   // GBK_TO_UNICODE[24568] := 16#C949;
   // GBK_TO_UNICODE[24569] := 16#848A;
   // GBK_TO_UNICODE[24570] := 16#C94A;
   // GBK_TO_UNICODE[24571] := 16#848D;
   // GBK_TO_UNICODE[24572] := 16#C94B;
   // GBK_TO_UNICODE[24573] := 16#848F;
   // GBK_TO_UNICODE[24574] := 16#C94C;
   // GBK_TO_UNICODE[24575] := 16#8490;
   // GBK_TO_UNICODE[24576] := 16#C94D;
   // GBK_TO_UNICODE[24577] := 16#8491;
   // GBK_TO_UNICODE[24578] := 16#C94E;
   // GBK_TO_UNICODE[24579] := 16#8492;
   // GBK_TO_UNICODE[24580] := 16#C94F;
   // GBK_TO_UNICODE[24581] := 16#8493;
   // GBK_TO_UNICODE[24582] := 16#C950;
   // GBK_TO_UNICODE[24583] := 16#8494;
   // GBK_TO_UNICODE[24584] := 16#C951;
   // GBK_TO_UNICODE[24585] := 16#8495;
   // GBK_TO_UNICODE[24586] := 16#C952;
   // GBK_TO_UNICODE[24587] := 16#8496;
   // GBK_TO_UNICODE[24588] := 16#C953;
   // GBK_TO_UNICODE[24589] := 16#8498;
   // GBK_TO_UNICODE[24590] := 16#C954;
   // GBK_TO_UNICODE[24591] := 16#849A;
   // GBK_TO_UNICODE[24592] := 16#C955;
   // GBK_TO_UNICODE[24593] := 16#849B;
   // GBK_TO_UNICODE[24594] := 16#C956;
   // GBK_TO_UNICODE[24595] := 16#849D;
   // GBK_TO_UNICODE[24596] := 16#C957;
   // GBK_TO_UNICODE[24597] := 16#849E;
   // GBK_TO_UNICODE[24598] := 16#C958;
   // GBK_TO_UNICODE[24599] := 16#849F;
   // GBK_TO_UNICODE[24600] := 16#C959;
   // GBK_TO_UNICODE[24601] := 16#84A0;
   // GBK_TO_UNICODE[24602] := 16#C95A;
   // GBK_TO_UNICODE[24603] := 16#84A2;
   // GBK_TO_UNICODE[24604] := 16#C95B;
   // GBK_TO_UNICODE[24605] := 16#84A3;
   // GBK_TO_UNICODE[24606] := 16#C95C;
   // GBK_TO_UNICODE[24607] := 16#84A4;
   // GBK_TO_UNICODE[24608] := 16#C95D;
   // GBK_TO_UNICODE[24609] := 16#84A5;
   // GBK_TO_UNICODE[24610] := 16#C95E;
   // GBK_TO_UNICODE[24611] := 16#84A6;
   // GBK_TO_UNICODE[24612] := 16#C95F;
   // GBK_TO_UNICODE[24613] := 16#84A7;
   // GBK_TO_UNICODE[24614] := 16#C960;
   // GBK_TO_UNICODE[24615] := 16#84A8;
   // GBK_TO_UNICODE[24616] := 16#C961;
   // GBK_TO_UNICODE[24617] := 16#84A9;
   // GBK_TO_UNICODE[24618] := 16#C962;
   // GBK_TO_UNICODE[24619] := 16#84AA;
   // GBK_TO_UNICODE[24620] := 16#C963;
   // GBK_TO_UNICODE[24621] := 16#84AB;
   // GBK_TO_UNICODE[24622] := 16#C964;
   // GBK_TO_UNICODE[24623] := 16#84AC;
   // GBK_TO_UNICODE[24624] := 16#C965;
   // GBK_TO_UNICODE[24625] := 16#84AD;
   // GBK_TO_UNICODE[24626] := 16#C966;
   // GBK_TO_UNICODE[24627] := 16#84AE;
   // GBK_TO_UNICODE[24628] := 16#C967;
   // GBK_TO_UNICODE[24629] := 16#84B0;
   // GBK_TO_UNICODE[24630] := 16#C968;
   // GBK_TO_UNICODE[24631] := 16#84B1;
   // GBK_TO_UNICODE[24632] := 16#C969;
   // GBK_TO_UNICODE[24633] := 16#84B3;
   // GBK_TO_UNICODE[24634] := 16#C96A;
   // GBK_TO_UNICODE[24635] := 16#84B5;
   // GBK_TO_UNICODE[24636] := 16#C96B;
   // GBK_TO_UNICODE[24637] := 16#84B6;
   // GBK_TO_UNICODE[24638] := 16#C96C;
   // GBK_TO_UNICODE[24639] := 16#84B7;
   // GBK_TO_UNICODE[24640] := 16#C96D;
   // GBK_TO_UNICODE[24641] := 16#84BB;
   // GBK_TO_UNICODE[24642] := 16#C96E;
   // GBK_TO_UNICODE[24643] := 16#84BC;
   // GBK_TO_UNICODE[24644] := 16#C96F;
   // GBK_TO_UNICODE[24645] := 16#84BE;
   // GBK_TO_UNICODE[24646] := 16#C970;
   // GBK_TO_UNICODE[24647] := 16#84C0;
   // GBK_TO_UNICODE[24648] := 16#C971;
   // GBK_TO_UNICODE[24649] := 16#84C2;
   // GBK_TO_UNICODE[24650] := 16#C972;
   // GBK_TO_UNICODE[24651] := 16#84C3;
   // GBK_TO_UNICODE[24652] := 16#C973;
   // GBK_TO_UNICODE[24653] := 16#84C5;
   // GBK_TO_UNICODE[24654] := 16#C974;
   // GBK_TO_UNICODE[24655] := 16#84C6;
   // GBK_TO_UNICODE[24656] := 16#C975;
   // GBK_TO_UNICODE[24657] := 16#84C7;
   // GBK_TO_UNICODE[24658] := 16#C976;
   // GBK_TO_UNICODE[24659] := 16#84C8;
   // GBK_TO_UNICODE[24660] := 16#C977;
   // GBK_TO_UNICODE[24661] := 16#84CB;
   // GBK_TO_UNICODE[24662] := 16#C978;
   // GBK_TO_UNICODE[24663] := 16#84CC;
   // GBK_TO_UNICODE[24664] := 16#C979;
   // GBK_TO_UNICODE[24665] := 16#84CE;
   // GBK_TO_UNICODE[24666] := 16#C97A;
   // GBK_TO_UNICODE[24667] := 16#84CF;
   // GBK_TO_UNICODE[24668] := 16#C97B;
   // GBK_TO_UNICODE[24669] := 16#84D2;
   // GBK_TO_UNICODE[24670] := 16#C97C;
   // GBK_TO_UNICODE[24671] := 16#84D4;
   // GBK_TO_UNICODE[24672] := 16#C97D;
   // GBK_TO_UNICODE[24673] := 16#84D5;
   // GBK_TO_UNICODE[24674] := 16#C97E;
   // GBK_TO_UNICODE[24675] := 16#84D7;
   // GBK_TO_UNICODE[24676] := 16#C980;
   // GBK_TO_UNICODE[24677] := 16#84D8;
   // GBK_TO_UNICODE[24678] := 16#C981;
   // GBK_TO_UNICODE[24679] := 16#84D9;
   // GBK_TO_UNICODE[24680] := 16#C982;
   // GBK_TO_UNICODE[24681] := 16#84DA;
   // GBK_TO_UNICODE[24682] := 16#C983;
   // GBK_TO_UNICODE[24683] := 16#84DB;
   // GBK_TO_UNICODE[24684] := 16#C984;
   // GBK_TO_UNICODE[24685] := 16#84DC;
   // GBK_TO_UNICODE[24686] := 16#C985;
   // GBK_TO_UNICODE[24687] := 16#84DE;
   // GBK_TO_UNICODE[24688] := 16#C986;
   // GBK_TO_UNICODE[24689] := 16#84E1;
   // GBK_TO_UNICODE[24690] := 16#C987;
   // GBK_TO_UNICODE[24691] := 16#84E2;
   // GBK_TO_UNICODE[24692] := 16#C988;
   // GBK_TO_UNICODE[24693] := 16#84E4;
   // GBK_TO_UNICODE[24694] := 16#C989;
   // GBK_TO_UNICODE[24695] := 16#84E7;
   // GBK_TO_UNICODE[24696] := 16#C98A;
   // GBK_TO_UNICODE[24697] := 16#84E8;
   // GBK_TO_UNICODE[24698] := 16#C98B;
   // GBK_TO_UNICODE[24699] := 16#84E9;
   // GBK_TO_UNICODE[24700] := 16#C98C;
   // GBK_TO_UNICODE[24701] := 16#84EA;
   // GBK_TO_UNICODE[24702] := 16#C98D;
   // GBK_TO_UNICODE[24703] := 16#84EB;
   // GBK_TO_UNICODE[24704] := 16#C98E;
   // GBK_TO_UNICODE[24705] := 16#84ED;
   // GBK_TO_UNICODE[24706] := 16#C98F;
   // GBK_TO_UNICODE[24707] := 16#84EE;
   // GBK_TO_UNICODE[24708] := 16#C990;
   // GBK_TO_UNICODE[24709] := 16#84EF;
   // GBK_TO_UNICODE[24710] := 16#C991;
   // GBK_TO_UNICODE[24711] := 16#84F1;
   // GBK_TO_UNICODE[24712] := 16#C992;
   // GBK_TO_UNICODE[24713] := 16#84F2;
   // GBK_TO_UNICODE[24714] := 16#C993;
   // GBK_TO_UNICODE[24715] := 16#84F3;
   // GBK_TO_UNICODE[24716] := 16#C994;
   // GBK_TO_UNICODE[24717] := 16#84F4;
   // GBK_TO_UNICODE[24718] := 16#C995;
   // GBK_TO_UNICODE[24719] := 16#84F5;
   // GBK_TO_UNICODE[24720] := 16#C996;
   // GBK_TO_UNICODE[24721] := 16#84F6;
   // GBK_TO_UNICODE[24722] := 16#C997;
   // GBK_TO_UNICODE[24723] := 16#84F7;
   // GBK_TO_UNICODE[24724] := 16#C998;
   // GBK_TO_UNICODE[24725] := 16#84F8;
   // GBK_TO_UNICODE[24726] := 16#C999;
   // GBK_TO_UNICODE[24727] := 16#84F9;
   // GBK_TO_UNICODE[24728] := 16#C99A;
   // GBK_TO_UNICODE[24729] := 16#84FA;
   // GBK_TO_UNICODE[24730] := 16#C99B;
   // GBK_TO_UNICODE[24731] := 16#84FB;
   // GBK_TO_UNICODE[24732] := 16#C99C;
   // GBK_TO_UNICODE[24733] := 16#84FD;
   // GBK_TO_UNICODE[24734] := 16#C99D;
   // GBK_TO_UNICODE[24735] := 16#84FE;
   // GBK_TO_UNICODE[24736] := 16#C99E;
   // GBK_TO_UNICODE[24737] := 16#8500;
   // GBK_TO_UNICODE[24738] := 16#C99F;
   // GBK_TO_UNICODE[24739] := 16#8501;
   // GBK_TO_UNICODE[24740] := 16#C9A0;
   // GBK_TO_UNICODE[24741] := 16#8502;
   // GBK_TO_UNICODE[24742] := 16#C9A1;
   // GBK_TO_UNICODE[24743] := 16#4F1E;
   // GBK_TO_UNICODE[24744] := 16#C9A2;
   // GBK_TO_UNICODE[24745] := 16#6563;
   // GBK_TO_UNICODE[24746] := 16#C9A3;
   // GBK_TO_UNICODE[24747] := 16#6851;
   // GBK_TO_UNICODE[24748] := 16#C9A4;
   // GBK_TO_UNICODE[24749] := 16#55D3;
   // GBK_TO_UNICODE[24750] := 16#C9A5;
   // GBK_TO_UNICODE[24751] := 16#4E27;
   // GBK_TO_UNICODE[24752] := 16#C9A6;
   // GBK_TO_UNICODE[24753] := 16#6414;
   // GBK_TO_UNICODE[24754] := 16#C9A7;
   // GBK_TO_UNICODE[24755] := 16#9A9A;
   // GBK_TO_UNICODE[24756] := 16#C9A8;
   // GBK_TO_UNICODE[24757] := 16#626B;
   // GBK_TO_UNICODE[24758] := 16#C9A9;
   // GBK_TO_UNICODE[24759] := 16#5AC2;
   // GBK_TO_UNICODE[24760] := 16#C9AA;
   // GBK_TO_UNICODE[24761] := 16#745F;
   // GBK_TO_UNICODE[24762] := 16#C9AB;
   // GBK_TO_UNICODE[24763] := 16#8272;
   // GBK_TO_UNICODE[24764] := 16#C9AC;
   // GBK_TO_UNICODE[24765] := 16#6DA9;
   // GBK_TO_UNICODE[24766] := 16#C9AD;
   // GBK_TO_UNICODE[24767] := 16#68EE;
   // GBK_TO_UNICODE[24768] := 16#C9AE;
   // GBK_TO_UNICODE[24769] := 16#50E7;
   // GBK_TO_UNICODE[24770] := 16#C9AF;
   // GBK_TO_UNICODE[24771] := 16#838E;
   // GBK_TO_UNICODE[24772] := 16#C9B0;
   // GBK_TO_UNICODE[24773] := 16#7802;
   // GBK_TO_UNICODE[24774] := 16#C9B1;
   // GBK_TO_UNICODE[24775] := 16#6740;
   // GBK_TO_UNICODE[24776] := 16#C9B2;
   // GBK_TO_UNICODE[24777] := 16#5239;
   // GBK_TO_UNICODE[24778] := 16#C9B3;
   // GBK_TO_UNICODE[24779] := 16#6C99;
   // GBK_TO_UNICODE[24780] := 16#C9B4;
   // GBK_TO_UNICODE[24781] := 16#7EB1;
   // GBK_TO_UNICODE[24782] := 16#C9B5;
   // GBK_TO_UNICODE[24783] := 16#50BB;
   // GBK_TO_UNICODE[24784] := 16#C9B6;
   // GBK_TO_UNICODE[24785] := 16#5565;
   // GBK_TO_UNICODE[24786] := 16#C9B7;
   // GBK_TO_UNICODE[24787] := 16#715E;
   // GBK_TO_UNICODE[24788] := 16#C9B8;
   // GBK_TO_UNICODE[24789] := 16#7B5B;
   // GBK_TO_UNICODE[24790] := 16#C9B9;
   // GBK_TO_UNICODE[24791] := 16#6652;
   // GBK_TO_UNICODE[24792] := 16#C9BA;
   // GBK_TO_UNICODE[24793] := 16#73CA;
   // GBK_TO_UNICODE[24794] := 16#C9BB;
   // GBK_TO_UNICODE[24795] := 16#82EB;
   // GBK_TO_UNICODE[24796] := 16#C9BC;
   // GBK_TO_UNICODE[24797] := 16#6749;
   // GBK_TO_UNICODE[24798] := 16#C9BD;
   // GBK_TO_UNICODE[24799] := 16#5C71;
   // GBK_TO_UNICODE[24800] := 16#C9BE;
   // GBK_TO_UNICODE[24801] := 16#5220;
   // GBK_TO_UNICODE[24802] := 16#C9BF;
   // GBK_TO_UNICODE[24803] := 16#717D;
   // GBK_TO_UNICODE[24804] := 16#C9C0;
   // GBK_TO_UNICODE[24805] := 16#886B;
   // GBK_TO_UNICODE[24806] := 16#C9C1;
   // GBK_TO_UNICODE[24807] := 16#95EA;
   // GBK_TO_UNICODE[24808] := 16#C9C2;
   // GBK_TO_UNICODE[24809] := 16#9655;
   // GBK_TO_UNICODE[24810] := 16#C9C3;
   // GBK_TO_UNICODE[24811] := 16#64C5;
   // GBK_TO_UNICODE[24812] := 16#C9C4;
   // GBK_TO_UNICODE[24813] := 16#8D61;
   // GBK_TO_UNICODE[24814] := 16#C9C5;
   // GBK_TO_UNICODE[24815] := 16#81B3;
   // GBK_TO_UNICODE[24816] := 16#C9C6;
   // GBK_TO_UNICODE[24817] := 16#5584;
   // GBK_TO_UNICODE[24818] := 16#C9C7;
   // GBK_TO_UNICODE[24819] := 16#6C55;
   // GBK_TO_UNICODE[24820] := 16#C9C8;
   // GBK_TO_UNICODE[24821] := 16#6247;
   // GBK_TO_UNICODE[24822] := 16#C9C9;
   // GBK_TO_UNICODE[24823] := 16#7F2E;
   // GBK_TO_UNICODE[24824] := 16#C9CA;
   // GBK_TO_UNICODE[24825] := 16#5892;
   // GBK_TO_UNICODE[24826] := 16#C9CB;
   // GBK_TO_UNICODE[24827] := 16#4F24;
   // GBK_TO_UNICODE[24828] := 16#C9CC;
   // GBK_TO_UNICODE[24829] := 16#5546;
   // GBK_TO_UNICODE[24830] := 16#C9CD;
   // GBK_TO_UNICODE[24831] := 16#8D4F;
   // GBK_TO_UNICODE[24832] := 16#C9CE;
   // GBK_TO_UNICODE[24833] := 16#664C;
   // GBK_TO_UNICODE[24834] := 16#C9CF;
   // GBK_TO_UNICODE[24835] := 16#4E0A;
   // GBK_TO_UNICODE[24836] := 16#C9D0;
   // GBK_TO_UNICODE[24837] := 16#5C1A;
   // GBK_TO_UNICODE[24838] := 16#C9D1;
   // GBK_TO_UNICODE[24839] := 16#88F3;
   // GBK_TO_UNICODE[24840] := 16#C9D2;
   // GBK_TO_UNICODE[24841] := 16#68A2;
   // GBK_TO_UNICODE[24842] := 16#C9D3;
   // GBK_TO_UNICODE[24843] := 16#634E;
   // GBK_TO_UNICODE[24844] := 16#C9D4;
   // GBK_TO_UNICODE[24845] := 16#7A0D;
   // GBK_TO_UNICODE[24846] := 16#C9D5;
   // GBK_TO_UNICODE[24847] := 16#70E7;
   // GBK_TO_UNICODE[24848] := 16#C9D6;
   // GBK_TO_UNICODE[24849] := 16#828D;
   // GBK_TO_UNICODE[24850] := 16#C9D7;
   // GBK_TO_UNICODE[24851] := 16#52FA;
   // GBK_TO_UNICODE[24852] := 16#C9D8;
   // GBK_TO_UNICODE[24853] := 16#97F6;
   // GBK_TO_UNICODE[24854] := 16#C9D9;
   // GBK_TO_UNICODE[24855] := 16#5C11;
   // GBK_TO_UNICODE[24856] := 16#C9DA;
   // GBK_TO_UNICODE[24857] := 16#54E8;
   // GBK_TO_UNICODE[24858] := 16#C9DB;
   // GBK_TO_UNICODE[24859] := 16#90B5;
   // GBK_TO_UNICODE[24860] := 16#C9DC;
   // GBK_TO_UNICODE[24861] := 16#7ECD;
   // GBK_TO_UNICODE[24862] := 16#C9DD;
   // GBK_TO_UNICODE[24863] := 16#5962;
   // GBK_TO_UNICODE[24864] := 16#C9DE;
   // GBK_TO_UNICODE[24865] := 16#8D4A;
   // GBK_TO_UNICODE[24866] := 16#C9DF;
   // GBK_TO_UNICODE[24867] := 16#86C7;
   // GBK_TO_UNICODE[24868] := 16#C9E0;
   // GBK_TO_UNICODE[24869] := 16#820C;
   // GBK_TO_UNICODE[24870] := 16#C9E1;
   // GBK_TO_UNICODE[24871] := 16#820D;
   // GBK_TO_UNICODE[24872] := 16#C9E2;
   // GBK_TO_UNICODE[24873] := 16#8D66;
   // GBK_TO_UNICODE[24874] := 16#C9E3;
   // GBK_TO_UNICODE[24875] := 16#6444;
   // GBK_TO_UNICODE[24876] := 16#C9E4;
   // GBK_TO_UNICODE[24877] := 16#5C04;
   // GBK_TO_UNICODE[24878] := 16#C9E5;
   // GBK_TO_UNICODE[24879] := 16#6151;
   // GBK_TO_UNICODE[24880] := 16#C9E6;
   // GBK_TO_UNICODE[24881] := 16#6D89;
   // GBK_TO_UNICODE[24882] := 16#C9E7;
   // GBK_TO_UNICODE[24883] := 16#793E;
   // GBK_TO_UNICODE[24884] := 16#C9E8;
   // GBK_TO_UNICODE[24885] := 16#8BBE;
   // GBK_TO_UNICODE[24886] := 16#C9E9;
   // GBK_TO_UNICODE[24887] := 16#7837;
   // GBK_TO_UNICODE[24888] := 16#C9EA;
   // GBK_TO_UNICODE[24889] := 16#7533;
   // GBK_TO_UNICODE[24890] := 16#C9EB;
   // GBK_TO_UNICODE[24891] := 16#547B;
   // GBK_TO_UNICODE[24892] := 16#C9EC;
   // GBK_TO_UNICODE[24893] := 16#4F38;
   // GBK_TO_UNICODE[24894] := 16#C9ED;
   // GBK_TO_UNICODE[24895] := 16#8EAB;
   // GBK_TO_UNICODE[24896] := 16#C9EE;
   // GBK_TO_UNICODE[24897] := 16#6DF1;
   // GBK_TO_UNICODE[24898] := 16#C9EF;
   // GBK_TO_UNICODE[24899] := 16#5A20;
   // GBK_TO_UNICODE[24900] := 16#C9F0;
   // GBK_TO_UNICODE[24901] := 16#7EC5;
   // GBK_TO_UNICODE[24902] := 16#C9F1;
   // GBK_TO_UNICODE[24903] := 16#795E;
   // GBK_TO_UNICODE[24904] := 16#C9F2;
   // GBK_TO_UNICODE[24905] := 16#6C88;
   // GBK_TO_UNICODE[24906] := 16#C9F3;
   // GBK_TO_UNICODE[24907] := 16#5BA1;
   // GBK_TO_UNICODE[24908] := 16#C9F4;
   // GBK_TO_UNICODE[24909] := 16#5A76;
   // GBK_TO_UNICODE[24910] := 16#C9F5;
   // GBK_TO_UNICODE[24911] := 16#751A;
   // GBK_TO_UNICODE[24912] := 16#C9F6;
   // GBK_TO_UNICODE[24913] := 16#80BE;
   // GBK_TO_UNICODE[24914] := 16#C9F7;
   // GBK_TO_UNICODE[24915] := 16#614E;
   // GBK_TO_UNICODE[24916] := 16#C9F8;
   // GBK_TO_UNICODE[24917] := 16#6E17;
   // GBK_TO_UNICODE[24918] := 16#C9F9;
   // GBK_TO_UNICODE[24919] := 16#58F0;
   // GBK_TO_UNICODE[24920] := 16#C9FA;
   // GBK_TO_UNICODE[24921] := 16#751F;
   // GBK_TO_UNICODE[24922] := 16#C9FB;
   // GBK_TO_UNICODE[24923] := 16#7525;
   // GBK_TO_UNICODE[24924] := 16#C9FC;
   // GBK_TO_UNICODE[24925] := 16#7272;
   // GBK_TO_UNICODE[24926] := 16#C9FD;
   // GBK_TO_UNICODE[24927] := 16#5347;
   // GBK_TO_UNICODE[24928] := 16#C9FE;
   // GBK_TO_UNICODE[24929] := 16#7EF3;
   // GBK_TO_UNICODE[24930] := 16#CA40;
   // GBK_TO_UNICODE[24931] := 16#8503;
   // GBK_TO_UNICODE[24932] := 16#CA41;
   // GBK_TO_UNICODE[24933] := 16#8504;
   // GBK_TO_UNICODE[24934] := 16#CA42;
   // GBK_TO_UNICODE[24935] := 16#8505;
   // GBK_TO_UNICODE[24936] := 16#CA43;
   // GBK_TO_UNICODE[24937] := 16#8506;
   // GBK_TO_UNICODE[24938] := 16#CA44;
   // GBK_TO_UNICODE[24939] := 16#8507;
   // GBK_TO_UNICODE[24940] := 16#CA45;
   // GBK_TO_UNICODE[24941] := 16#8508;
   // GBK_TO_UNICODE[24942] := 16#CA46;
   // GBK_TO_UNICODE[24943] := 16#8509;
   // GBK_TO_UNICODE[24944] := 16#CA47;
   // GBK_TO_UNICODE[24945] := 16#850A;
   // GBK_TO_UNICODE[24946] := 16#CA48;
   // GBK_TO_UNICODE[24947] := 16#850B;
   // GBK_TO_UNICODE[24948] := 16#CA49;
   // GBK_TO_UNICODE[24949] := 16#850D;
   // GBK_TO_UNICODE[24950] := 16#CA4A;
   // GBK_TO_UNICODE[24951] := 16#850E;
   // GBK_TO_UNICODE[24952] := 16#CA4B;
   // GBK_TO_UNICODE[24953] := 16#850F;
   // GBK_TO_UNICODE[24954] := 16#CA4C;
   // GBK_TO_UNICODE[24955] := 16#8510;
   // GBK_TO_UNICODE[24956] := 16#CA4D;
   // GBK_TO_UNICODE[24957] := 16#8512;
   // GBK_TO_UNICODE[24958] := 16#CA4E;
   // GBK_TO_UNICODE[24959] := 16#8514;
   // GBK_TO_UNICODE[24960] := 16#CA4F;
   // GBK_TO_UNICODE[24961] := 16#8515;
   // GBK_TO_UNICODE[24962] := 16#CA50;
   // GBK_TO_UNICODE[24963] := 16#8516;
   // GBK_TO_UNICODE[24964] := 16#CA51;
   // GBK_TO_UNICODE[24965] := 16#8518;
   // GBK_TO_UNICODE[24966] := 16#CA52;
   // GBK_TO_UNICODE[24967] := 16#8519;
   // GBK_TO_UNICODE[24968] := 16#CA53;
   // GBK_TO_UNICODE[24969] := 16#851B;
   // GBK_TO_UNICODE[24970] := 16#CA54;
   // GBK_TO_UNICODE[24971] := 16#851C;
   // GBK_TO_UNICODE[24972] := 16#CA55;
   // GBK_TO_UNICODE[24973] := 16#851D;
   // GBK_TO_UNICODE[24974] := 16#CA56;
   // GBK_TO_UNICODE[24975] := 16#851E;
   // GBK_TO_UNICODE[24976] := 16#CA57;
   // GBK_TO_UNICODE[24977] := 16#8520;
   // GBK_TO_UNICODE[24978] := 16#CA58;
   // GBK_TO_UNICODE[24979] := 16#8522;
   // GBK_TO_UNICODE[24980] := 16#CA59;
   // GBK_TO_UNICODE[24981] := 16#8523;
   // GBK_TO_UNICODE[24982] := 16#CA5A;
   // GBK_TO_UNICODE[24983] := 16#8524;
   // GBK_TO_UNICODE[24984] := 16#CA5B;
   // GBK_TO_UNICODE[24985] := 16#8525;
   // GBK_TO_UNICODE[24986] := 16#CA5C;
   // GBK_TO_UNICODE[24987] := 16#8526;
   // GBK_TO_UNICODE[24988] := 16#CA5D;
   // GBK_TO_UNICODE[24989] := 16#8527;
   // GBK_TO_UNICODE[24990] := 16#CA5E;
   // GBK_TO_UNICODE[24991] := 16#8528;
   // GBK_TO_UNICODE[24992] := 16#CA5F;
   // GBK_TO_UNICODE[24993] := 16#8529;
   // GBK_TO_UNICODE[24994] := 16#CA60;
   // GBK_TO_UNICODE[24995] := 16#852A;
   // GBK_TO_UNICODE[24996] := 16#CA61;
   // GBK_TO_UNICODE[24997] := 16#852D;
   // GBK_TO_UNICODE[24998] := 16#CA62;
   // GBK_TO_UNICODE[24999] := 16#852E;
   // GBK_TO_UNICODE[25000] := 16#CA63;
   // GBK_TO_UNICODE[25001] := 16#852F;
   // GBK_TO_UNICODE[25002] := 16#CA64;
   // GBK_TO_UNICODE[25003] := 16#8530;
   // GBK_TO_UNICODE[25004] := 16#CA65;
   // GBK_TO_UNICODE[25005] := 16#8531;
   // GBK_TO_UNICODE[25006] := 16#CA66;
   // GBK_TO_UNICODE[25007] := 16#8532;
   // GBK_TO_UNICODE[25008] := 16#CA67;
   // GBK_TO_UNICODE[25009] := 16#8533;
   // GBK_TO_UNICODE[25010] := 16#CA68;
   // GBK_TO_UNICODE[25011] := 16#8534;
   // GBK_TO_UNICODE[25012] := 16#CA69;
   // GBK_TO_UNICODE[25013] := 16#8535;
   // GBK_TO_UNICODE[25014] := 16#CA6A;
   // GBK_TO_UNICODE[25015] := 16#8536;
   // GBK_TO_UNICODE[25016] := 16#CA6B;
   // GBK_TO_UNICODE[25017] := 16#853E;
   // GBK_TO_UNICODE[25018] := 16#CA6C;
   // GBK_TO_UNICODE[25019] := 16#853F;
   // GBK_TO_UNICODE[25020] := 16#CA6D;
   // GBK_TO_UNICODE[25021] := 16#8540;
   // GBK_TO_UNICODE[25022] := 16#CA6E;
   // GBK_TO_UNICODE[25023] := 16#8541;
   // GBK_TO_UNICODE[25024] := 16#CA6F;
   // GBK_TO_UNICODE[25025] := 16#8542;
   // GBK_TO_UNICODE[25026] := 16#CA70;
   // GBK_TO_UNICODE[25027] := 16#8544;
   // GBK_TO_UNICODE[25028] := 16#CA71;
   // GBK_TO_UNICODE[25029] := 16#8545;
   // GBK_TO_UNICODE[25030] := 16#CA72;
   // GBK_TO_UNICODE[25031] := 16#8546;
   // GBK_TO_UNICODE[25032] := 16#CA73;
   // GBK_TO_UNICODE[25033] := 16#8547;
   // GBK_TO_UNICODE[25034] := 16#CA74;
   // GBK_TO_UNICODE[25035] := 16#854B;
   // GBK_TO_UNICODE[25036] := 16#CA75;
   // GBK_TO_UNICODE[25037] := 16#854C;
   // GBK_TO_UNICODE[25038] := 16#CA76;
   // GBK_TO_UNICODE[25039] := 16#854D;
   // GBK_TO_UNICODE[25040] := 16#CA77;
   // GBK_TO_UNICODE[25041] := 16#854E;
   // GBK_TO_UNICODE[25042] := 16#CA78;
   // GBK_TO_UNICODE[25043] := 16#854F;
   // GBK_TO_UNICODE[25044] := 16#CA79;
   // GBK_TO_UNICODE[25045] := 16#8550;
   // GBK_TO_UNICODE[25046] := 16#CA7A;
   // GBK_TO_UNICODE[25047] := 16#8551;
   // GBK_TO_UNICODE[25048] := 16#CA7B;
   // GBK_TO_UNICODE[25049] := 16#8552;
   // GBK_TO_UNICODE[25050] := 16#CA7C;
   // GBK_TO_UNICODE[25051] := 16#8553;
   // GBK_TO_UNICODE[25052] := 16#CA7D;
   // GBK_TO_UNICODE[25053] := 16#8554;
   // GBK_TO_UNICODE[25054] := 16#CA7E;
   // GBK_TO_UNICODE[25055] := 16#8555;
   // GBK_TO_UNICODE[25056] := 16#CA80;
   // GBK_TO_UNICODE[25057] := 16#8557;
   // GBK_TO_UNICODE[25058] := 16#CA81;
   // GBK_TO_UNICODE[25059] := 16#8558;
   // GBK_TO_UNICODE[25060] := 16#CA82;
   // GBK_TO_UNICODE[25061] := 16#855A;
   // GBK_TO_UNICODE[25062] := 16#CA83;
   // GBK_TO_UNICODE[25063] := 16#855B;
   // GBK_TO_UNICODE[25064] := 16#CA84;
   // GBK_TO_UNICODE[25065] := 16#855C;
   // GBK_TO_UNICODE[25066] := 16#CA85;
   // GBK_TO_UNICODE[25067] := 16#855D;
   // GBK_TO_UNICODE[25068] := 16#CA86;
   // GBK_TO_UNICODE[25069] := 16#855F;
   // GBK_TO_UNICODE[25070] := 16#CA87;
   // GBK_TO_UNICODE[25071] := 16#8560;
   // GBK_TO_UNICODE[25072] := 16#CA88;
   // GBK_TO_UNICODE[25073] := 16#8561;
   // GBK_TO_UNICODE[25074] := 16#CA89;
   // GBK_TO_UNICODE[25075] := 16#8562;
   // GBK_TO_UNICODE[25076] := 16#CA8A;
   // GBK_TO_UNICODE[25077] := 16#8563;
   // GBK_TO_UNICODE[25078] := 16#CA8B;
   // GBK_TO_UNICODE[25079] := 16#8565;
   // GBK_TO_UNICODE[25080] := 16#CA8C;
   // GBK_TO_UNICODE[25081] := 16#8566;
   // GBK_TO_UNICODE[25082] := 16#CA8D;
   // GBK_TO_UNICODE[25083] := 16#8567;
   // GBK_TO_UNICODE[25084] := 16#CA8E;
   // GBK_TO_UNICODE[25085] := 16#8569;
   // GBK_TO_UNICODE[25086] := 16#CA8F;
   // GBK_TO_UNICODE[25087] := 16#856A;
   // GBK_TO_UNICODE[25088] := 16#CA90;
   // GBK_TO_UNICODE[25089] := 16#856B;
   // GBK_TO_UNICODE[25090] := 16#CA91;
   // GBK_TO_UNICODE[25091] := 16#856C;
   // GBK_TO_UNICODE[25092] := 16#CA92;
   // GBK_TO_UNICODE[25093] := 16#856D;
   // GBK_TO_UNICODE[25094] := 16#CA93;
   // GBK_TO_UNICODE[25095] := 16#856E;
   // GBK_TO_UNICODE[25096] := 16#CA94;
   // GBK_TO_UNICODE[25097] := 16#856F;
   // GBK_TO_UNICODE[25098] := 16#CA95;
   // GBK_TO_UNICODE[25099] := 16#8570;
   // GBK_TO_UNICODE[25100] := 16#CA96;
   // GBK_TO_UNICODE[25101] := 16#8571;
   // GBK_TO_UNICODE[25102] := 16#CA97;
   // GBK_TO_UNICODE[25103] := 16#8573;
   // GBK_TO_UNICODE[25104] := 16#CA98;
   // GBK_TO_UNICODE[25105] := 16#8575;
   // GBK_TO_UNICODE[25106] := 16#CA99;
   // GBK_TO_UNICODE[25107] := 16#8576;
   // GBK_TO_UNICODE[25108] := 16#CA9A;
   // GBK_TO_UNICODE[25109] := 16#8577;
   // GBK_TO_UNICODE[25110] := 16#CA9B;
   // GBK_TO_UNICODE[25111] := 16#8578;
   // GBK_TO_UNICODE[25112] := 16#CA9C;
   // GBK_TO_UNICODE[25113] := 16#857C;
   // GBK_TO_UNICODE[25114] := 16#CA9D;
   // GBK_TO_UNICODE[25115] := 16#857D;
   // GBK_TO_UNICODE[25116] := 16#CA9E;
   // GBK_TO_UNICODE[25117] := 16#857F;
   // GBK_TO_UNICODE[25118] := 16#CA9F;
   // GBK_TO_UNICODE[25119] := 16#8580;
   // GBK_TO_UNICODE[25120] := 16#CAA0;
   // GBK_TO_UNICODE[25121] := 16#8581;
   // GBK_TO_UNICODE[25122] := 16#CAA1;
   // GBK_TO_UNICODE[25123] := 16#7701;
   // GBK_TO_UNICODE[25124] := 16#CAA2;
   // GBK_TO_UNICODE[25125] := 16#76DB;
   // GBK_TO_UNICODE[25126] := 16#CAA3;
   // GBK_TO_UNICODE[25127] := 16#5269;
   // GBK_TO_UNICODE[25128] := 16#CAA4;
   // GBK_TO_UNICODE[25129] := 16#80DC;
   // GBK_TO_UNICODE[25130] := 16#CAA5;
   // GBK_TO_UNICODE[25131] := 16#5723;
   // GBK_TO_UNICODE[25132] := 16#CAA6;
   // GBK_TO_UNICODE[25133] := 16#5E08;
   // GBK_TO_UNICODE[25134] := 16#CAA7;
   // GBK_TO_UNICODE[25135] := 16#5931;
   // GBK_TO_UNICODE[25136] := 16#CAA8;
   // GBK_TO_UNICODE[25137] := 16#72EE;
   // GBK_TO_UNICODE[25138] := 16#CAA9;
   // GBK_TO_UNICODE[25139] := 16#65BD;
   // GBK_TO_UNICODE[25140] := 16#CAAA;
   // GBK_TO_UNICODE[25141] := 16#6E7F;
   // GBK_TO_UNICODE[25142] := 16#CAAB;
   // GBK_TO_UNICODE[25143] := 16#8BD7;
   // GBK_TO_UNICODE[25144] := 16#CAAC;
   // GBK_TO_UNICODE[25145] := 16#5C38;
   // GBK_TO_UNICODE[25146] := 16#CAAD;
   // GBK_TO_UNICODE[25147] := 16#8671;
   // GBK_TO_UNICODE[25148] := 16#CAAE;
   // GBK_TO_UNICODE[25149] := 16#5341;
   // GBK_TO_UNICODE[25150] := 16#CAAF;
   // GBK_TO_UNICODE[25151] := 16#77F3;
   // GBK_TO_UNICODE[25152] := 16#CAB0;
   // GBK_TO_UNICODE[25153] := 16#62FE;
   // GBK_TO_UNICODE[25154] := 16#CAB1;
   // GBK_TO_UNICODE[25155] := 16#65F6;
   // GBK_TO_UNICODE[25156] := 16#CAB2;
   // GBK_TO_UNICODE[25157] := 16#4EC0;
   // GBK_TO_UNICODE[25158] := 16#CAB3;
   // GBK_TO_UNICODE[25159] := 16#98DF;
   // GBK_TO_UNICODE[25160] := 16#CAB4;
   // GBK_TO_UNICODE[25161] := 16#8680;
   // GBK_TO_UNICODE[25162] := 16#CAB5;
   // GBK_TO_UNICODE[25163] := 16#5B9E;
   // GBK_TO_UNICODE[25164] := 16#CAB6;
   // GBK_TO_UNICODE[25165] := 16#8BC6;
   // GBK_TO_UNICODE[25166] := 16#CAB7;
   // GBK_TO_UNICODE[25167] := 16#53F2;
   // GBK_TO_UNICODE[25168] := 16#CAB8;
   // GBK_TO_UNICODE[25169] := 16#77E2;
   // GBK_TO_UNICODE[25170] := 16#CAB9;
   // GBK_TO_UNICODE[25171] := 16#4F7F;
   // GBK_TO_UNICODE[25172] := 16#CABA;
   // GBK_TO_UNICODE[25173] := 16#5C4E;
   // GBK_TO_UNICODE[25174] := 16#CABB;
   // GBK_TO_UNICODE[25175] := 16#9A76;
   // GBK_TO_UNICODE[25176] := 16#CABC;
   // GBK_TO_UNICODE[25177] := 16#59CB;
   // GBK_TO_UNICODE[25178] := 16#CABD;
   // GBK_TO_UNICODE[25179] := 16#5F0F;
   // GBK_TO_UNICODE[25180] := 16#CABE;
   // GBK_TO_UNICODE[25181] := 16#793A;
   // GBK_TO_UNICODE[25182] := 16#CABF;
   // GBK_TO_UNICODE[25183] := 16#58EB;
   // GBK_TO_UNICODE[25184] := 16#CAC0;
   // GBK_TO_UNICODE[25185] := 16#4E16;
   // GBK_TO_UNICODE[25186] := 16#CAC1;
   // GBK_TO_UNICODE[25187] := 16#67FF;
   // GBK_TO_UNICODE[25188] := 16#CAC2;
   // GBK_TO_UNICODE[25189] := 16#4E8B;
   // GBK_TO_UNICODE[25190] := 16#CAC3;
   // GBK_TO_UNICODE[25191] := 16#62ED;
   // GBK_TO_UNICODE[25192] := 16#CAC4;
   // GBK_TO_UNICODE[25193] := 16#8A93;
   // GBK_TO_UNICODE[25194] := 16#CAC5;
   // GBK_TO_UNICODE[25195] := 16#901D;
   // GBK_TO_UNICODE[25196] := 16#CAC6;
   // GBK_TO_UNICODE[25197] := 16#52BF;
   // GBK_TO_UNICODE[25198] := 16#CAC7;
   // GBK_TO_UNICODE[25199] := 16#662F;
   // GBK_TO_UNICODE[25200] := 16#CAC8;
   // GBK_TO_UNICODE[25201] := 16#55DC;
   // GBK_TO_UNICODE[25202] := 16#CAC9;
   // GBK_TO_UNICODE[25203] := 16#566C;
   // GBK_TO_UNICODE[25204] := 16#CACA;
   // GBK_TO_UNICODE[25205] := 16#9002;
   // GBK_TO_UNICODE[25206] := 16#CACB;
   // GBK_TO_UNICODE[25207] := 16#4ED5;
   // GBK_TO_UNICODE[25208] := 16#CACC;
   // GBK_TO_UNICODE[25209] := 16#4F8D;
   // GBK_TO_UNICODE[25210] := 16#CACD;
   // GBK_TO_UNICODE[25211] := 16#91CA;
   // GBK_TO_UNICODE[25212] := 16#CACE;
   // GBK_TO_UNICODE[25213] := 16#9970;
   // GBK_TO_UNICODE[25214] := 16#CACF;
   // GBK_TO_UNICODE[25215] := 16#6C0F;
   // GBK_TO_UNICODE[25216] := 16#CAD0;
   // GBK_TO_UNICODE[25217] := 16#5E02;
   // GBK_TO_UNICODE[25218] := 16#CAD1;
   // GBK_TO_UNICODE[25219] := 16#6043;
   // GBK_TO_UNICODE[25220] := 16#CAD2;
   // GBK_TO_UNICODE[25221] := 16#5BA4;
   // GBK_TO_UNICODE[25222] := 16#CAD3;
   // GBK_TO_UNICODE[25223] := 16#89C6;
   // GBK_TO_UNICODE[25224] := 16#CAD4;
   // GBK_TO_UNICODE[25225] := 16#8BD5;
   // GBK_TO_UNICODE[25226] := 16#CAD5;
   // GBK_TO_UNICODE[25227] := 16#6536;
   // GBK_TO_UNICODE[25228] := 16#CAD6;
   // GBK_TO_UNICODE[25229] := 16#624B;
   // GBK_TO_UNICODE[25230] := 16#CAD7;
   // GBK_TO_UNICODE[25231] := 16#9996;
   // GBK_TO_UNICODE[25232] := 16#CAD8;
   // GBK_TO_UNICODE[25233] := 16#5B88;
   // GBK_TO_UNICODE[25234] := 16#CAD9;
   // GBK_TO_UNICODE[25235] := 16#5BFF;
   // GBK_TO_UNICODE[25236] := 16#CADA;
   // GBK_TO_UNICODE[25237] := 16#6388;
   // GBK_TO_UNICODE[25238] := 16#CADB;
   // GBK_TO_UNICODE[25239] := 16#552E;
   // GBK_TO_UNICODE[25240] := 16#CADC;
   // GBK_TO_UNICODE[25241] := 16#53D7;
   // GBK_TO_UNICODE[25242] := 16#CADD;
   // GBK_TO_UNICODE[25243] := 16#7626;
   // GBK_TO_UNICODE[25244] := 16#CADE;
   // GBK_TO_UNICODE[25245] := 16#517D;
   // GBK_TO_UNICODE[25246] := 16#CADF;
   // GBK_TO_UNICODE[25247] := 16#852C;
   // GBK_TO_UNICODE[25248] := 16#CAE0;
   // GBK_TO_UNICODE[25249] := 16#67A2;
   // GBK_TO_UNICODE[25250] := 16#CAE1;
   // GBK_TO_UNICODE[25251] := 16#68B3;
   // GBK_TO_UNICODE[25252] := 16#CAE2;
   // GBK_TO_UNICODE[25253] := 16#6B8A;
   // GBK_TO_UNICODE[25254] := 16#CAE3;
   // GBK_TO_UNICODE[25255] := 16#6292;
   // GBK_TO_UNICODE[25256] := 16#CAE4;
   // GBK_TO_UNICODE[25257] := 16#8F93;
   // GBK_TO_UNICODE[25258] := 16#CAE5;
   // GBK_TO_UNICODE[25259] := 16#53D4;
   // GBK_TO_UNICODE[25260] := 16#CAE6;
   // GBK_TO_UNICODE[25261] := 16#8212;
   // GBK_TO_UNICODE[25262] := 16#CAE7;
   // GBK_TO_UNICODE[25263] := 16#6DD1;
   // GBK_TO_UNICODE[25264] := 16#CAE8;
   // GBK_TO_UNICODE[25265] := 16#758F;
   // GBK_TO_UNICODE[25266] := 16#CAE9;
   // GBK_TO_UNICODE[25267] := 16#4E66;
   // GBK_TO_UNICODE[25268] := 16#CAEA;
   // GBK_TO_UNICODE[25269] := 16#8D4E;
   // GBK_TO_UNICODE[25270] := 16#CAEB;
   // GBK_TO_UNICODE[25271] := 16#5B70;
   // GBK_TO_UNICODE[25272] := 16#CAEC;
   // GBK_TO_UNICODE[25273] := 16#719F;
   // GBK_TO_UNICODE[25274] := 16#CAED;
   // GBK_TO_UNICODE[25275] := 16#85AF;
   // GBK_TO_UNICODE[25276] := 16#CAEE;
   // GBK_TO_UNICODE[25277] := 16#6691;
   // GBK_TO_UNICODE[25278] := 16#CAEF;
   // GBK_TO_UNICODE[25279] := 16#66D9;
   // GBK_TO_UNICODE[25280] := 16#CAF0;
   // GBK_TO_UNICODE[25281] := 16#7F72;
   // GBK_TO_UNICODE[25282] := 16#CAF1;
   // GBK_TO_UNICODE[25283] := 16#8700;
   // GBK_TO_UNICODE[25284] := 16#CAF2;
   // GBK_TO_UNICODE[25285] := 16#9ECD;
   // GBK_TO_UNICODE[25286] := 16#CAF3;
   // GBK_TO_UNICODE[25287] := 16#9F20;
   // GBK_TO_UNICODE[25288] := 16#CAF4;
   // GBK_TO_UNICODE[25289] := 16#5C5E;
   // GBK_TO_UNICODE[25290] := 16#CAF5;
   // GBK_TO_UNICODE[25291] := 16#672F;
   // GBK_TO_UNICODE[25292] := 16#CAF6;
   // GBK_TO_UNICODE[25293] := 16#8FF0;
   // GBK_TO_UNICODE[25294] := 16#CAF7;
   // GBK_TO_UNICODE[25295] := 16#6811;
   // GBK_TO_UNICODE[25296] := 16#CAF8;
   // GBK_TO_UNICODE[25297] := 16#675F;
   // GBK_TO_UNICODE[25298] := 16#CAF9;
   // GBK_TO_UNICODE[25299] := 16#620D;
   // GBK_TO_UNICODE[25300] := 16#CAFA;
   // GBK_TO_UNICODE[25301] := 16#7AD6;
   // GBK_TO_UNICODE[25302] := 16#CAFB;
   // GBK_TO_UNICODE[25303] := 16#5885;
   // GBK_TO_UNICODE[25304] := 16#CAFC;
   // GBK_TO_UNICODE[25305] := 16#5EB6;
   // GBK_TO_UNICODE[25306] := 16#CAFD;
   // GBK_TO_UNICODE[25307] := 16#6570;
   // GBK_TO_UNICODE[25308] := 16#CAFE;
   // GBK_TO_UNICODE[25309] := 16#6F31;
   // GBK_TO_UNICODE[25310] := 16#CB40;
   // GBK_TO_UNICODE[25311] := 16#8582;
   // GBK_TO_UNICODE[25312] := 16#CB41;
   // GBK_TO_UNICODE[25313] := 16#8583;
   // GBK_TO_UNICODE[25314] := 16#CB42;
   // GBK_TO_UNICODE[25315] := 16#8586;
   // GBK_TO_UNICODE[25316] := 16#CB43;
   // GBK_TO_UNICODE[25317] := 16#8588;
   // GBK_TO_UNICODE[25318] := 16#CB44;
   // GBK_TO_UNICODE[25319] := 16#8589;
   // GBK_TO_UNICODE[25320] := 16#CB45;
   // GBK_TO_UNICODE[25321] := 16#858A;
   // GBK_TO_UNICODE[25322] := 16#CB46;
   // GBK_TO_UNICODE[25323] := 16#858B;
   // GBK_TO_UNICODE[25324] := 16#CB47;
   // GBK_TO_UNICODE[25325] := 16#858C;
   // GBK_TO_UNICODE[25326] := 16#CB48;
   // GBK_TO_UNICODE[25327] := 16#858D;
   // GBK_TO_UNICODE[25328] := 16#CB49;
   // GBK_TO_UNICODE[25329] := 16#858E;
   // GBK_TO_UNICODE[25330] := 16#CB4A;
   // GBK_TO_UNICODE[25331] := 16#8590;
   // GBK_TO_UNICODE[25332] := 16#CB4B;
   // GBK_TO_UNICODE[25333] := 16#8591;
   // GBK_TO_UNICODE[25334] := 16#CB4C;
   // GBK_TO_UNICODE[25335] := 16#8592;
   // GBK_TO_UNICODE[25336] := 16#CB4D;
   // GBK_TO_UNICODE[25337] := 16#8593;
   // GBK_TO_UNICODE[25338] := 16#CB4E;
   // GBK_TO_UNICODE[25339] := 16#8594;
   // GBK_TO_UNICODE[25340] := 16#CB4F;
   // GBK_TO_UNICODE[25341] := 16#8595;
   // GBK_TO_UNICODE[25342] := 16#CB50;
   // GBK_TO_UNICODE[25343] := 16#8596;
   // GBK_TO_UNICODE[25344] := 16#CB51;
   // GBK_TO_UNICODE[25345] := 16#8597;
   // GBK_TO_UNICODE[25346] := 16#CB52;
   // GBK_TO_UNICODE[25347] := 16#8598;
   // GBK_TO_UNICODE[25348] := 16#CB53;
   // GBK_TO_UNICODE[25349] := 16#8599;
   // GBK_TO_UNICODE[25350] := 16#CB54;
   // GBK_TO_UNICODE[25351] := 16#859A;
   // GBK_TO_UNICODE[25352] := 16#CB55;
   // GBK_TO_UNICODE[25353] := 16#859D;
   // GBK_TO_UNICODE[25354] := 16#CB56;
   // GBK_TO_UNICODE[25355] := 16#859E;
   // GBK_TO_UNICODE[25356] := 16#CB57;
   // GBK_TO_UNICODE[25357] := 16#859F;
   // GBK_TO_UNICODE[25358] := 16#CB58;
   // GBK_TO_UNICODE[25359] := 16#85A0;
   // GBK_TO_UNICODE[25360] := 16#CB59;
   // GBK_TO_UNICODE[25361] := 16#85A1;
   // GBK_TO_UNICODE[25362] := 16#CB5A;
   // GBK_TO_UNICODE[25363] := 16#85A2;
   // GBK_TO_UNICODE[25364] := 16#CB5B;
   // GBK_TO_UNICODE[25365] := 16#85A3;
   // GBK_TO_UNICODE[25366] := 16#CB5C;
   // GBK_TO_UNICODE[25367] := 16#85A5;
   // GBK_TO_UNICODE[25368] := 16#CB5D;
   // GBK_TO_UNICODE[25369] := 16#85A6;
   // GBK_TO_UNICODE[25370] := 16#CB5E;
   // GBK_TO_UNICODE[25371] := 16#85A7;
   // GBK_TO_UNICODE[25372] := 16#CB5F;
   // GBK_TO_UNICODE[25373] := 16#85A9;
   // GBK_TO_UNICODE[25374] := 16#CB60;
   // GBK_TO_UNICODE[25375] := 16#85AB;
   // GBK_TO_UNICODE[25376] := 16#CB61;
   // GBK_TO_UNICODE[25377] := 16#85AC;
   // GBK_TO_UNICODE[25378] := 16#CB62;
   // GBK_TO_UNICODE[25379] := 16#85AD;
   // GBK_TO_UNICODE[25380] := 16#CB63;
   // GBK_TO_UNICODE[25381] := 16#85B1;
   // GBK_TO_UNICODE[25382] := 16#CB64;
   // GBK_TO_UNICODE[25383] := 16#85B2;
   // GBK_TO_UNICODE[25384] := 16#CB65;
   // GBK_TO_UNICODE[25385] := 16#85B3;
   // GBK_TO_UNICODE[25386] := 16#CB66;
   // GBK_TO_UNICODE[25387] := 16#85B4;
   // GBK_TO_UNICODE[25388] := 16#CB67;
   // GBK_TO_UNICODE[25389] := 16#85B5;
   // GBK_TO_UNICODE[25390] := 16#CB68;
   // GBK_TO_UNICODE[25391] := 16#85B6;
   // GBK_TO_UNICODE[25392] := 16#CB69;
   // GBK_TO_UNICODE[25393] := 16#85B8;
   // GBK_TO_UNICODE[25394] := 16#CB6A;
   // GBK_TO_UNICODE[25395] := 16#85BA;
   // GBK_TO_UNICODE[25396] := 16#CB6B;
   // GBK_TO_UNICODE[25397] := 16#85BB;
   // GBK_TO_UNICODE[25398] := 16#CB6C;
   // GBK_TO_UNICODE[25399] := 16#85BC;
   // GBK_TO_UNICODE[25400] := 16#CB6D;
   // GBK_TO_UNICODE[25401] := 16#85BD;
   // GBK_TO_UNICODE[25402] := 16#CB6E;
   // GBK_TO_UNICODE[25403] := 16#85BE;
   // GBK_TO_UNICODE[25404] := 16#CB6F;
   // GBK_TO_UNICODE[25405] := 16#85BF;
   // GBK_TO_UNICODE[25406] := 16#CB70;
   // GBK_TO_UNICODE[25407] := 16#85C0;
   // GBK_TO_UNICODE[25408] := 16#CB71;
   // GBK_TO_UNICODE[25409] := 16#85C2;
   // GBK_TO_UNICODE[25410] := 16#CB72;
   // GBK_TO_UNICODE[25411] := 16#85C3;
   // GBK_TO_UNICODE[25412] := 16#CB73;
   // GBK_TO_UNICODE[25413] := 16#85C4;
   // GBK_TO_UNICODE[25414] := 16#CB74;
   // GBK_TO_UNICODE[25415] := 16#85C5;
   // GBK_TO_UNICODE[25416] := 16#CB75;
   // GBK_TO_UNICODE[25417] := 16#85C6;
   // GBK_TO_UNICODE[25418] := 16#CB76;
   // GBK_TO_UNICODE[25419] := 16#85C7;
   // GBK_TO_UNICODE[25420] := 16#CB77;
   // GBK_TO_UNICODE[25421] := 16#85C8;
   // GBK_TO_UNICODE[25422] := 16#CB78;
   // GBK_TO_UNICODE[25423] := 16#85CA;
   // GBK_TO_UNICODE[25424] := 16#CB79;
   // GBK_TO_UNICODE[25425] := 16#85CB;
   // GBK_TO_UNICODE[25426] := 16#CB7A;
   // GBK_TO_UNICODE[25427] := 16#85CC;
   // GBK_TO_UNICODE[25428] := 16#CB7B;
   // GBK_TO_UNICODE[25429] := 16#85CD;
   // GBK_TO_UNICODE[25430] := 16#CB7C;
   // GBK_TO_UNICODE[25431] := 16#85CE;
   // GBK_TO_UNICODE[25432] := 16#CB7D;
   // GBK_TO_UNICODE[25433] := 16#85D1;
   // GBK_TO_UNICODE[25434] := 16#CB7E;
   // GBK_TO_UNICODE[25435] := 16#85D2;
   // GBK_TO_UNICODE[25436] := 16#CB80;
   // GBK_TO_UNICODE[25437] := 16#85D4;
   // GBK_TO_UNICODE[25438] := 16#CB81;
   // GBK_TO_UNICODE[25439] := 16#85D6;
   // GBK_TO_UNICODE[25440] := 16#CB82;
   // GBK_TO_UNICODE[25441] := 16#85D7;
   // GBK_TO_UNICODE[25442] := 16#CB83;
   // GBK_TO_UNICODE[25443] := 16#85D8;
   // GBK_TO_UNICODE[25444] := 16#CB84;
   // GBK_TO_UNICODE[25445] := 16#85D9;
   // GBK_TO_UNICODE[25446] := 16#CB85;
   // GBK_TO_UNICODE[25447] := 16#85DA;
   // GBK_TO_UNICODE[25448] := 16#CB86;
   // GBK_TO_UNICODE[25449] := 16#85DB;
   // GBK_TO_UNICODE[25450] := 16#CB87;
   // GBK_TO_UNICODE[25451] := 16#85DD;
   // GBK_TO_UNICODE[25452] := 16#CB88;
   // GBK_TO_UNICODE[25453] := 16#85DE;
   // GBK_TO_UNICODE[25454] := 16#CB89;
   // GBK_TO_UNICODE[25455] := 16#85DF;
   // GBK_TO_UNICODE[25456] := 16#CB8A;
   // GBK_TO_UNICODE[25457] := 16#85E0;
   // GBK_TO_UNICODE[25458] := 16#CB8B;
   // GBK_TO_UNICODE[25459] := 16#85E1;
   // GBK_TO_UNICODE[25460] := 16#CB8C;
   // GBK_TO_UNICODE[25461] := 16#85E2;
   // GBK_TO_UNICODE[25462] := 16#CB8D;
   // GBK_TO_UNICODE[25463] := 16#85E3;
   // GBK_TO_UNICODE[25464] := 16#CB8E;
   // GBK_TO_UNICODE[25465] := 16#85E5;
   // GBK_TO_UNICODE[25466] := 16#CB8F;
   // GBK_TO_UNICODE[25467] := 16#85E6;
   // GBK_TO_UNICODE[25468] := 16#CB90;
   // GBK_TO_UNICODE[25469] := 16#85E7;
   // GBK_TO_UNICODE[25470] := 16#CB91;
   // GBK_TO_UNICODE[25471] := 16#85E8;
   // GBK_TO_UNICODE[25472] := 16#CB92;
   // GBK_TO_UNICODE[25473] := 16#85EA;
   // GBK_TO_UNICODE[25474] := 16#CB93;
   // GBK_TO_UNICODE[25475] := 16#85EB;
   // GBK_TO_UNICODE[25476] := 16#CB94;
   // GBK_TO_UNICODE[25477] := 16#85EC;
   // GBK_TO_UNICODE[25478] := 16#CB95;
   // GBK_TO_UNICODE[25479] := 16#85ED;
   // GBK_TO_UNICODE[25480] := 16#CB96;
   // GBK_TO_UNICODE[25481] := 16#85EE;
   // GBK_TO_UNICODE[25482] := 16#CB97;
   // GBK_TO_UNICODE[25483] := 16#85EF;
   // GBK_TO_UNICODE[25484] := 16#CB98;
   // GBK_TO_UNICODE[25485] := 16#85F0;
   // GBK_TO_UNICODE[25486] := 16#CB99;
   // GBK_TO_UNICODE[25487] := 16#85F1;
   // GBK_TO_UNICODE[25488] := 16#CB9A;
   // GBK_TO_UNICODE[25489] := 16#85F2;
   // GBK_TO_UNICODE[25490] := 16#CB9B;
   // GBK_TO_UNICODE[25491] := 16#85F3;
   // GBK_TO_UNICODE[25492] := 16#CB9C;
   // GBK_TO_UNICODE[25493] := 16#85F4;
   // GBK_TO_UNICODE[25494] := 16#CB9D;
   // GBK_TO_UNICODE[25495] := 16#85F5;
   // GBK_TO_UNICODE[25496] := 16#CB9E;
   // GBK_TO_UNICODE[25497] := 16#85F6;
   // GBK_TO_UNICODE[25498] := 16#CB9F;
   // GBK_TO_UNICODE[25499] := 16#85F7;
   // GBK_TO_UNICODE[25500] := 16#CBA0;
   // GBK_TO_UNICODE[25501] := 16#85F8;
   // GBK_TO_UNICODE[25502] := 16#CBA1;
   // GBK_TO_UNICODE[25503] := 16#6055;
   // GBK_TO_UNICODE[25504] := 16#CBA2;
   // GBK_TO_UNICODE[25505] := 16#5237;
   // GBK_TO_UNICODE[25506] := 16#CBA3;
   // GBK_TO_UNICODE[25507] := 16#800D;
   // GBK_TO_UNICODE[25508] := 16#CBA4;
   // GBK_TO_UNICODE[25509] := 16#6454;
   // GBK_TO_UNICODE[25510] := 16#CBA5;
   // GBK_TO_UNICODE[25511] := 16#8870;
   // GBK_TO_UNICODE[25512] := 16#CBA6;
   // GBK_TO_UNICODE[25513] := 16#7529;
   // GBK_TO_UNICODE[25514] := 16#CBA7;
   // GBK_TO_UNICODE[25515] := 16#5E05;
   // GBK_TO_UNICODE[25516] := 16#CBA8;
   // GBK_TO_UNICODE[25517] := 16#6813;
   // GBK_TO_UNICODE[25518] := 16#CBA9;
   // GBK_TO_UNICODE[25519] := 16#62F4;
   // GBK_TO_UNICODE[25520] := 16#CBAA;
   // GBK_TO_UNICODE[25521] := 16#971C;
   // GBK_TO_UNICODE[25522] := 16#CBAB;
   // GBK_TO_UNICODE[25523] := 16#53CC;
   // GBK_TO_UNICODE[25524] := 16#CBAC;
   // GBK_TO_UNICODE[25525] := 16#723D;
   // GBK_TO_UNICODE[25526] := 16#CBAD;
   // GBK_TO_UNICODE[25527] := 16#8C01;
   // GBK_TO_UNICODE[25528] := 16#CBAE;
   // GBK_TO_UNICODE[25529] := 16#6C34;
   // GBK_TO_UNICODE[25530] := 16#CBAF;
   // GBK_TO_UNICODE[25531] := 16#7761;
   // GBK_TO_UNICODE[25532] := 16#CBB0;
   // GBK_TO_UNICODE[25533] := 16#7A0E;
   // GBK_TO_UNICODE[25534] := 16#CBB1;
   // GBK_TO_UNICODE[25535] := 16#542E;
   // GBK_TO_UNICODE[25536] := 16#CBB2;
   // GBK_TO_UNICODE[25537] := 16#77AC;
   // GBK_TO_UNICODE[25538] := 16#CBB3;
   // GBK_TO_UNICODE[25539] := 16#987A;
   // GBK_TO_UNICODE[25540] := 16#CBB4;
   // GBK_TO_UNICODE[25541] := 16#821C;
   // GBK_TO_UNICODE[25542] := 16#CBB5;
   // GBK_TO_UNICODE[25543] := 16#8BF4;
   // GBK_TO_UNICODE[25544] := 16#CBB6;
   // GBK_TO_UNICODE[25545] := 16#7855;
   // GBK_TO_UNICODE[25546] := 16#CBB7;
   // GBK_TO_UNICODE[25547] := 16#6714;
   // GBK_TO_UNICODE[25548] := 16#CBB8;
   // GBK_TO_UNICODE[25549] := 16#70C1;
   // GBK_TO_UNICODE[25550] := 16#CBB9;
   // GBK_TO_UNICODE[25551] := 16#65AF;
   // GBK_TO_UNICODE[25552] := 16#CBBA;
   // GBK_TO_UNICODE[25553] := 16#6495;
   // GBK_TO_UNICODE[25554] := 16#CBBB;
   // GBK_TO_UNICODE[25555] := 16#5636;
   // GBK_TO_UNICODE[25556] := 16#CBBC;
   // GBK_TO_UNICODE[25557] := 16#601D;
   // GBK_TO_UNICODE[25558] := 16#CBBD;
   // GBK_TO_UNICODE[25559] := 16#79C1;
   // GBK_TO_UNICODE[25560] := 16#CBBE;
   // GBK_TO_UNICODE[25561] := 16#53F8;
   // GBK_TO_UNICODE[25562] := 16#CBBF;
   // GBK_TO_UNICODE[25563] := 16#4E1D;
   // GBK_TO_UNICODE[25564] := 16#CBC0;
   // GBK_TO_UNICODE[25565] := 16#6B7B;
   // GBK_TO_UNICODE[25566] := 16#CBC1;
   // GBK_TO_UNICODE[25567] := 16#8086;
   // GBK_TO_UNICODE[25568] := 16#CBC2;
   // GBK_TO_UNICODE[25569] := 16#5BFA;
   // GBK_TO_UNICODE[25570] := 16#CBC3;
   // GBK_TO_UNICODE[25571] := 16#55E3;
   // GBK_TO_UNICODE[25572] := 16#CBC4;
   // GBK_TO_UNICODE[25573] := 16#56DB;
   // GBK_TO_UNICODE[25574] := 16#CBC5;
   // GBK_TO_UNICODE[25575] := 16#4F3A;
   // GBK_TO_UNICODE[25576] := 16#CBC6;
   // GBK_TO_UNICODE[25577] := 16#4F3C;
   // GBK_TO_UNICODE[25578] := 16#CBC7;
   // GBK_TO_UNICODE[25579] := 16#9972;
   // GBK_TO_UNICODE[25580] := 16#CBC8;
   // GBK_TO_UNICODE[25581] := 16#5DF3;
   // GBK_TO_UNICODE[25582] := 16#CBC9;
   // GBK_TO_UNICODE[25583] := 16#677E;
   // GBK_TO_UNICODE[25584] := 16#CBCA;
   // GBK_TO_UNICODE[25585] := 16#8038;
   // GBK_TO_UNICODE[25586] := 16#CBCB;
   // GBK_TO_UNICODE[25587] := 16#6002;
   // GBK_TO_UNICODE[25588] := 16#CBCC;
   // GBK_TO_UNICODE[25589] := 16#9882;
   // GBK_TO_UNICODE[25590] := 16#CBCD;
   // GBK_TO_UNICODE[25591] := 16#9001;
   // GBK_TO_UNICODE[25592] := 16#CBCE;
   // GBK_TO_UNICODE[25593] := 16#5B8B;
   // GBK_TO_UNICODE[25594] := 16#CBCF;
   // GBK_TO_UNICODE[25595] := 16#8BBC;
   // GBK_TO_UNICODE[25596] := 16#CBD0;
   // GBK_TO_UNICODE[25597] := 16#8BF5;
   // GBK_TO_UNICODE[25598] := 16#CBD1;
   // GBK_TO_UNICODE[25599] := 16#641C;
   // GBK_TO_UNICODE[25600] := 16#CBD2;
   // GBK_TO_UNICODE[25601] := 16#8258;
   // GBK_TO_UNICODE[25602] := 16#CBD3;
   // GBK_TO_UNICODE[25603] := 16#64DE;
   // GBK_TO_UNICODE[25604] := 16#CBD4;
   // GBK_TO_UNICODE[25605] := 16#55FD;
   // GBK_TO_UNICODE[25606] := 16#CBD5;
   // GBK_TO_UNICODE[25607] := 16#82CF;
   // GBK_TO_UNICODE[25608] := 16#CBD6;
   // GBK_TO_UNICODE[25609] := 16#9165;
   // GBK_TO_UNICODE[25610] := 16#CBD7;
   // GBK_TO_UNICODE[25611] := 16#4FD7;
   // GBK_TO_UNICODE[25612] := 16#CBD8;
   // GBK_TO_UNICODE[25613] := 16#7D20;
   // GBK_TO_UNICODE[25614] := 16#CBD9;
   // GBK_TO_UNICODE[25615] := 16#901F;
   // GBK_TO_UNICODE[25616] := 16#CBDA;
   // GBK_TO_UNICODE[25617] := 16#7C9F;
   // GBK_TO_UNICODE[25618] := 16#CBDB;
   // GBK_TO_UNICODE[25619] := 16#50F3;
   // GBK_TO_UNICODE[25620] := 16#CBDC;
   // GBK_TO_UNICODE[25621] := 16#5851;
   // GBK_TO_UNICODE[25622] := 16#CBDD;
   // GBK_TO_UNICODE[25623] := 16#6EAF;
   // GBK_TO_UNICODE[25624] := 16#CBDE;
   // GBK_TO_UNICODE[25625] := 16#5BBF;
   // GBK_TO_UNICODE[25626] := 16#CBDF;
   // GBK_TO_UNICODE[25627] := 16#8BC9;
   // GBK_TO_UNICODE[25628] := 16#CBE0;
   // GBK_TO_UNICODE[25629] := 16#8083;
   // GBK_TO_UNICODE[25630] := 16#CBE1;
   // GBK_TO_UNICODE[25631] := 16#9178;
   // GBK_TO_UNICODE[25632] := 16#CBE2;
   // GBK_TO_UNICODE[25633] := 16#849C;
   // GBK_TO_UNICODE[25634] := 16#CBE3;
   // GBK_TO_UNICODE[25635] := 16#7B97;
   // GBK_TO_UNICODE[25636] := 16#CBE4;
   // GBK_TO_UNICODE[25637] := 16#867D;
   // GBK_TO_UNICODE[25638] := 16#CBE5;
   // GBK_TO_UNICODE[25639] := 16#968B;
   // GBK_TO_UNICODE[25640] := 16#CBE6;
   // GBK_TO_UNICODE[25641] := 16#968F;
   // GBK_TO_UNICODE[25642] := 16#CBE7;
   // GBK_TO_UNICODE[25643] := 16#7EE5;
   // GBK_TO_UNICODE[25644] := 16#CBE8;
   // GBK_TO_UNICODE[25645] := 16#9AD3;
   // GBK_TO_UNICODE[25646] := 16#CBE9;
   // GBK_TO_UNICODE[25647] := 16#788E;
   // GBK_TO_UNICODE[25648] := 16#CBEA;
   // GBK_TO_UNICODE[25649] := 16#5C81;
   // GBK_TO_UNICODE[25650] := 16#CBEB;
   // GBK_TO_UNICODE[25651] := 16#7A57;
   // GBK_TO_UNICODE[25652] := 16#CBEC;
   // GBK_TO_UNICODE[25653] := 16#9042;
   // GBK_TO_UNICODE[25654] := 16#CBED;
   // GBK_TO_UNICODE[25655] := 16#96A7;
   // GBK_TO_UNICODE[25656] := 16#CBEE;
   // GBK_TO_UNICODE[25657] := 16#795F;
   // GBK_TO_UNICODE[25658] := 16#CBEF;
   // GBK_TO_UNICODE[25659] := 16#5B59;
   // GBK_TO_UNICODE[25660] := 16#CBF0;
   // GBK_TO_UNICODE[25661] := 16#635F;
   // GBK_TO_UNICODE[25662] := 16#CBF1;
   // GBK_TO_UNICODE[25663] := 16#7B0B;
   // GBK_TO_UNICODE[25664] := 16#CBF2;
   // GBK_TO_UNICODE[25665] := 16#84D1;
   // GBK_TO_UNICODE[25666] := 16#CBF3;
   // GBK_TO_UNICODE[25667] := 16#68AD;
   // GBK_TO_UNICODE[25668] := 16#CBF4;
   // GBK_TO_UNICODE[25669] := 16#5506;
   // GBK_TO_UNICODE[25670] := 16#CBF5;
   // GBK_TO_UNICODE[25671] := 16#7F29;
   // GBK_TO_UNICODE[25672] := 16#CBF6;
   // GBK_TO_UNICODE[25673] := 16#7410;
   // GBK_TO_UNICODE[25674] := 16#CBF7;
   // GBK_TO_UNICODE[25675] := 16#7D22;
   // GBK_TO_UNICODE[25676] := 16#CBF8;
   // GBK_TO_UNICODE[25677] := 16#9501;
   // GBK_TO_UNICODE[25678] := 16#CBF9;
   // GBK_TO_UNICODE[25679] := 16#6240;
   // GBK_TO_UNICODE[25680] := 16#CBFA;
   // GBK_TO_UNICODE[25681] := 16#584C;
   // GBK_TO_UNICODE[25682] := 16#CBFB;
   // GBK_TO_UNICODE[25683] := 16#4ED6;
   // GBK_TO_UNICODE[25684] := 16#CBFC;
   // GBK_TO_UNICODE[25685] := 16#5B83;
   // GBK_TO_UNICODE[25686] := 16#CBFD;
   // GBK_TO_UNICODE[25687] := 16#5979;
   // GBK_TO_UNICODE[25688] := 16#CBFE;
   // GBK_TO_UNICODE[25689] := 16#5854;
   // GBK_TO_UNICODE[25690] := 16#CC40;
   // GBK_TO_UNICODE[25691] := 16#85F9;
   // GBK_TO_UNICODE[25692] := 16#CC41;
   // GBK_TO_UNICODE[25693] := 16#85FA;
   // GBK_TO_UNICODE[25694] := 16#CC42;
   // GBK_TO_UNICODE[25695] := 16#85FC;
   // GBK_TO_UNICODE[25696] := 16#CC43;
   // GBK_TO_UNICODE[25697] := 16#85FD;
   // GBK_TO_UNICODE[25698] := 16#CC44;
   // GBK_TO_UNICODE[25699] := 16#85FE;
   // GBK_TO_UNICODE[25700] := 16#CC45;
   // GBK_TO_UNICODE[25701] := 16#8600;
   // GBK_TO_UNICODE[25702] := 16#CC46;
   // GBK_TO_UNICODE[25703] := 16#8601;
   // GBK_TO_UNICODE[25704] := 16#CC47;
   // GBK_TO_UNICODE[25705] := 16#8602;
   // GBK_TO_UNICODE[25706] := 16#CC48;
   // GBK_TO_UNICODE[25707] := 16#8603;
   // GBK_TO_UNICODE[25708] := 16#CC49;
   // GBK_TO_UNICODE[25709] := 16#8604;
   // GBK_TO_UNICODE[25710] := 16#CC4A;
   // GBK_TO_UNICODE[25711] := 16#8606;
   // GBK_TO_UNICODE[25712] := 16#CC4B;
   // GBK_TO_UNICODE[25713] := 16#8607;
   // GBK_TO_UNICODE[25714] := 16#CC4C;
   // GBK_TO_UNICODE[25715] := 16#8608;
   // GBK_TO_UNICODE[25716] := 16#CC4D;
   // GBK_TO_UNICODE[25717] := 16#8609;
   // GBK_TO_UNICODE[25718] := 16#CC4E;
   // GBK_TO_UNICODE[25719] := 16#860A;
   // GBK_TO_UNICODE[25720] := 16#CC4F;
   // GBK_TO_UNICODE[25721] := 16#860B;
   // GBK_TO_UNICODE[25722] := 16#CC50;
   // GBK_TO_UNICODE[25723] := 16#860C;
   // GBK_TO_UNICODE[25724] := 16#CC51;
   // GBK_TO_UNICODE[25725] := 16#860D;
   // GBK_TO_UNICODE[25726] := 16#CC52;
   // GBK_TO_UNICODE[25727] := 16#860E;
   // GBK_TO_UNICODE[25728] := 16#CC53;
   // GBK_TO_UNICODE[25729] := 16#860F;
   // GBK_TO_UNICODE[25730] := 16#CC54;
   // GBK_TO_UNICODE[25731] := 16#8610;
   // GBK_TO_UNICODE[25732] := 16#CC55;
   // GBK_TO_UNICODE[25733] := 16#8612;
   // GBK_TO_UNICODE[25734] := 16#CC56;
   // GBK_TO_UNICODE[25735] := 16#8613;
   // GBK_TO_UNICODE[25736] := 16#CC57;
   // GBK_TO_UNICODE[25737] := 16#8614;
   // GBK_TO_UNICODE[25738] := 16#CC58;
   // GBK_TO_UNICODE[25739] := 16#8615;
   // GBK_TO_UNICODE[25740] := 16#CC59;
   // GBK_TO_UNICODE[25741] := 16#8617;
   // GBK_TO_UNICODE[25742] := 16#CC5A;
   // GBK_TO_UNICODE[25743] := 16#8618;
   // GBK_TO_UNICODE[25744] := 16#CC5B;
   // GBK_TO_UNICODE[25745] := 16#8619;
   // GBK_TO_UNICODE[25746] := 16#CC5C;
   // GBK_TO_UNICODE[25747] := 16#861A;
   // GBK_TO_UNICODE[25748] := 16#CC5D;
   // GBK_TO_UNICODE[25749] := 16#861B;
   // GBK_TO_UNICODE[25750] := 16#CC5E;
   // GBK_TO_UNICODE[25751] := 16#861C;
   // GBK_TO_UNICODE[25752] := 16#CC5F;
   // GBK_TO_UNICODE[25753] := 16#861D;
   // GBK_TO_UNICODE[25754] := 16#CC60;
   // GBK_TO_UNICODE[25755] := 16#861E;
   // GBK_TO_UNICODE[25756] := 16#CC61;
   // GBK_TO_UNICODE[25757] := 16#861F;
   // GBK_TO_UNICODE[25758] := 16#CC62;
   // GBK_TO_UNICODE[25759] := 16#8620;
   // GBK_TO_UNICODE[25760] := 16#CC63;
   // GBK_TO_UNICODE[25761] := 16#8621;
   // GBK_TO_UNICODE[25762] := 16#CC64;
   // GBK_TO_UNICODE[25763] := 16#8622;
   // GBK_TO_UNICODE[25764] := 16#CC65;
   // GBK_TO_UNICODE[25765] := 16#8623;
   // GBK_TO_UNICODE[25766] := 16#CC66;
   // GBK_TO_UNICODE[25767] := 16#8624;
   // GBK_TO_UNICODE[25768] := 16#CC67;
   // GBK_TO_UNICODE[25769] := 16#8625;
   // GBK_TO_UNICODE[25770] := 16#CC68;
   // GBK_TO_UNICODE[25771] := 16#8626;
   // GBK_TO_UNICODE[25772] := 16#CC69;
   // GBK_TO_UNICODE[25773] := 16#8628;
   // GBK_TO_UNICODE[25774] := 16#CC6A;
   // GBK_TO_UNICODE[25775] := 16#862A;
   // GBK_TO_UNICODE[25776] := 16#CC6B;
   // GBK_TO_UNICODE[25777] := 16#862B;
   // GBK_TO_UNICODE[25778] := 16#CC6C;
   // GBK_TO_UNICODE[25779] := 16#862C;
   // GBK_TO_UNICODE[25780] := 16#CC6D;
   // GBK_TO_UNICODE[25781] := 16#862D;
   // GBK_TO_UNICODE[25782] := 16#CC6E;
   // GBK_TO_UNICODE[25783] := 16#862E;
   // GBK_TO_UNICODE[25784] := 16#CC6F;
   // GBK_TO_UNICODE[25785] := 16#862F;
   // GBK_TO_UNICODE[25786] := 16#CC70;
   // GBK_TO_UNICODE[25787] := 16#8630;
   // GBK_TO_UNICODE[25788] := 16#CC71;
   // GBK_TO_UNICODE[25789] := 16#8631;
   // GBK_TO_UNICODE[25790] := 16#CC72;
   // GBK_TO_UNICODE[25791] := 16#8632;
   // GBK_TO_UNICODE[25792] := 16#CC73;
   // GBK_TO_UNICODE[25793] := 16#8633;
   // GBK_TO_UNICODE[25794] := 16#CC74;
   // GBK_TO_UNICODE[25795] := 16#8634;
   // GBK_TO_UNICODE[25796] := 16#CC75;
   // GBK_TO_UNICODE[25797] := 16#8635;
   // GBK_TO_UNICODE[25798] := 16#CC76;
   // GBK_TO_UNICODE[25799] := 16#8636;
   // GBK_TO_UNICODE[25800] := 16#CC77;
   // GBK_TO_UNICODE[25801] := 16#8637;
   // GBK_TO_UNICODE[25802] := 16#CC78;
   // GBK_TO_UNICODE[25803] := 16#8639;
   // GBK_TO_UNICODE[25804] := 16#CC79;
   // GBK_TO_UNICODE[25805] := 16#863A;
   // GBK_TO_UNICODE[25806] := 16#CC7A;
   // GBK_TO_UNICODE[25807] := 16#863B;
   // GBK_TO_UNICODE[25808] := 16#CC7B;
   // GBK_TO_UNICODE[25809] := 16#863D;
   // GBK_TO_UNICODE[25810] := 16#CC7C;
   // GBK_TO_UNICODE[25811] := 16#863E;
   // GBK_TO_UNICODE[25812] := 16#CC7D;
   // GBK_TO_UNICODE[25813] := 16#863F;
   // GBK_TO_UNICODE[25814] := 16#CC7E;
   // GBK_TO_UNICODE[25815] := 16#8640;
   // GBK_TO_UNICODE[25816] := 16#CC80;
   // GBK_TO_UNICODE[25817] := 16#8641;
   // GBK_TO_UNICODE[25818] := 16#CC81;
   // GBK_TO_UNICODE[25819] := 16#8642;
   // GBK_TO_UNICODE[25820] := 16#CC82;
   // GBK_TO_UNICODE[25821] := 16#8643;
   // GBK_TO_UNICODE[25822] := 16#CC83;
   // GBK_TO_UNICODE[25823] := 16#8644;
   // GBK_TO_UNICODE[25824] := 16#CC84;
   // GBK_TO_UNICODE[25825] := 16#8645;
   // GBK_TO_UNICODE[25826] := 16#CC85;
   // GBK_TO_UNICODE[25827] := 16#8646;
   // GBK_TO_UNICODE[25828] := 16#CC86;
   // GBK_TO_UNICODE[25829] := 16#8647;
   // GBK_TO_UNICODE[25830] := 16#CC87;
   // GBK_TO_UNICODE[25831] := 16#8648;
   // GBK_TO_UNICODE[25832] := 16#CC88;
   // GBK_TO_UNICODE[25833] := 16#8649;
   // GBK_TO_UNICODE[25834] := 16#CC89;
   // GBK_TO_UNICODE[25835] := 16#864A;
   // GBK_TO_UNICODE[25836] := 16#CC8A;
   // GBK_TO_UNICODE[25837] := 16#864B;
   // GBK_TO_UNICODE[25838] := 16#CC8B;
   // GBK_TO_UNICODE[25839] := 16#864C;
   // GBK_TO_UNICODE[25840] := 16#CC8C;
   // GBK_TO_UNICODE[25841] := 16#8652;
   // GBK_TO_UNICODE[25842] := 16#CC8D;
   // GBK_TO_UNICODE[25843] := 16#8653;
   // GBK_TO_UNICODE[25844] := 16#CC8E;
   // GBK_TO_UNICODE[25845] := 16#8655;
   // GBK_TO_UNICODE[25846] := 16#CC8F;
   // GBK_TO_UNICODE[25847] := 16#8656;
   // GBK_TO_UNICODE[25848] := 16#CC90;
   // GBK_TO_UNICODE[25849] := 16#8657;
   // GBK_TO_UNICODE[25850] := 16#CC91;
   // GBK_TO_UNICODE[25851] := 16#8658;
   // GBK_TO_UNICODE[25852] := 16#CC92;
   // GBK_TO_UNICODE[25853] := 16#8659;
   // GBK_TO_UNICODE[25854] := 16#CC93;
   // GBK_TO_UNICODE[25855] := 16#865B;
   // GBK_TO_UNICODE[25856] := 16#CC94;
   // GBK_TO_UNICODE[25857] := 16#865C;
   // GBK_TO_UNICODE[25858] := 16#CC95;
   // GBK_TO_UNICODE[25859] := 16#865D;
   // GBK_TO_UNICODE[25860] := 16#CC96;
   // GBK_TO_UNICODE[25861] := 16#865F;
   // GBK_TO_UNICODE[25862] := 16#CC97;
   // GBK_TO_UNICODE[25863] := 16#8660;
   // GBK_TO_UNICODE[25864] := 16#CC98;
   // GBK_TO_UNICODE[25865] := 16#8661;
   // GBK_TO_UNICODE[25866] := 16#CC99;
   // GBK_TO_UNICODE[25867] := 16#8663;
   // GBK_TO_UNICODE[25868] := 16#CC9A;
   // GBK_TO_UNICODE[25869] := 16#8664;
   // GBK_TO_UNICODE[25870] := 16#CC9B;
   // GBK_TO_UNICODE[25871] := 16#8665;
   // GBK_TO_UNICODE[25872] := 16#CC9C;
   // GBK_TO_UNICODE[25873] := 16#8666;
   // GBK_TO_UNICODE[25874] := 16#CC9D;
   // GBK_TO_UNICODE[25875] := 16#8667;
   // GBK_TO_UNICODE[25876] := 16#CC9E;
   // GBK_TO_UNICODE[25877] := 16#8668;
   // GBK_TO_UNICODE[25878] := 16#CC9F;
   // GBK_TO_UNICODE[25879] := 16#8669;
   // GBK_TO_UNICODE[25880] := 16#CCA0;
   // GBK_TO_UNICODE[25881] := 16#866A;
   // GBK_TO_UNICODE[25882] := 16#CCA1;
   // GBK_TO_UNICODE[25883] := 16#736D;
   // GBK_TO_UNICODE[25884] := 16#CCA2;
   // GBK_TO_UNICODE[25885] := 16#631E;
   // GBK_TO_UNICODE[25886] := 16#CCA3;
   // GBK_TO_UNICODE[25887] := 16#8E4B;
   // GBK_TO_UNICODE[25888] := 16#CCA4;
   // GBK_TO_UNICODE[25889] := 16#8E0F;
   // GBK_TO_UNICODE[25890] := 16#CCA5;
   // GBK_TO_UNICODE[25891] := 16#80CE;
   // GBK_TO_UNICODE[25892] := 16#CCA6;
   // GBK_TO_UNICODE[25893] := 16#82D4;
   // GBK_TO_UNICODE[25894] := 16#CCA7;
   // GBK_TO_UNICODE[25895] := 16#62AC;
   // GBK_TO_UNICODE[25896] := 16#CCA8;
   // GBK_TO_UNICODE[25897] := 16#53F0;
   // GBK_TO_UNICODE[25898] := 16#CCA9;
   // GBK_TO_UNICODE[25899] := 16#6CF0;
   // GBK_TO_UNICODE[25900] := 16#CCAA;
   // GBK_TO_UNICODE[25901] := 16#915E;
   // GBK_TO_UNICODE[25902] := 16#CCAB;
   // GBK_TO_UNICODE[25903] := 16#592A;
   // GBK_TO_UNICODE[25904] := 16#CCAC;
   // GBK_TO_UNICODE[25905] := 16#6001;
   // GBK_TO_UNICODE[25906] := 16#CCAD;
   // GBK_TO_UNICODE[25907] := 16#6C70;
   // GBK_TO_UNICODE[25908] := 16#CCAE;
   // GBK_TO_UNICODE[25909] := 16#574D;
   // GBK_TO_UNICODE[25910] := 16#CCAF;
   // GBK_TO_UNICODE[25911] := 16#644A;
   // GBK_TO_UNICODE[25912] := 16#CCB0;
   // GBK_TO_UNICODE[25913] := 16#8D2A;
   // GBK_TO_UNICODE[25914] := 16#CCB1;
   // GBK_TO_UNICODE[25915] := 16#762B;
   // GBK_TO_UNICODE[25916] := 16#CCB2;
   // GBK_TO_UNICODE[25917] := 16#6EE9;
   // GBK_TO_UNICODE[25918] := 16#CCB3;
   // GBK_TO_UNICODE[25919] := 16#575B;
   // GBK_TO_UNICODE[25920] := 16#CCB4;
   // GBK_TO_UNICODE[25921] := 16#6A80;
   // GBK_TO_UNICODE[25922] := 16#CCB5;
   // GBK_TO_UNICODE[25923] := 16#75F0;
   // GBK_TO_UNICODE[25924] := 16#CCB6;
   // GBK_TO_UNICODE[25925] := 16#6F6D;
   // GBK_TO_UNICODE[25926] := 16#CCB7;
   // GBK_TO_UNICODE[25927] := 16#8C2D;
   // GBK_TO_UNICODE[25928] := 16#CCB8;
   // GBK_TO_UNICODE[25929] := 16#8C08;
   // GBK_TO_UNICODE[25930] := 16#CCB9;
   // GBK_TO_UNICODE[25931] := 16#5766;
   // GBK_TO_UNICODE[25932] := 16#CCBA;
   // GBK_TO_UNICODE[25933] := 16#6BEF;
   // GBK_TO_UNICODE[25934] := 16#CCBB;
   // GBK_TO_UNICODE[25935] := 16#8892;
   // GBK_TO_UNICODE[25936] := 16#CCBC;
   // GBK_TO_UNICODE[25937] := 16#78B3;
   // GBK_TO_UNICODE[25938] := 16#CCBD;
   // GBK_TO_UNICODE[25939] := 16#63A2;
   // GBK_TO_UNICODE[25940] := 16#CCBE;
   // GBK_TO_UNICODE[25941] := 16#53F9;
   // GBK_TO_UNICODE[25942] := 16#CCBF;
   // GBK_TO_UNICODE[25943] := 16#70AD;
   // GBK_TO_UNICODE[25944] := 16#CCC0;
   // GBK_TO_UNICODE[25945] := 16#6C64;
   // GBK_TO_UNICODE[25946] := 16#CCC1;
   // GBK_TO_UNICODE[25947] := 16#5858;
   // GBK_TO_UNICODE[25948] := 16#CCC2;
   // GBK_TO_UNICODE[25949] := 16#642A;
   // GBK_TO_UNICODE[25950] := 16#CCC3;
   // GBK_TO_UNICODE[25951] := 16#5802;
   // GBK_TO_UNICODE[25952] := 16#CCC4;
   // GBK_TO_UNICODE[25953] := 16#68E0;
   // GBK_TO_UNICODE[25954] := 16#CCC5;
   // GBK_TO_UNICODE[25955] := 16#819B;
   // GBK_TO_UNICODE[25956] := 16#CCC6;
   // GBK_TO_UNICODE[25957] := 16#5510;
   // GBK_TO_UNICODE[25958] := 16#CCC7;
   // GBK_TO_UNICODE[25959] := 16#7CD6;
   // GBK_TO_UNICODE[25960] := 16#CCC8;
   // GBK_TO_UNICODE[25961] := 16#5018;
   // GBK_TO_UNICODE[25962] := 16#CCC9;
   // GBK_TO_UNICODE[25963] := 16#8EBA;
   // GBK_TO_UNICODE[25964] := 16#CCCA;
   // GBK_TO_UNICODE[25965] := 16#6DCC;
   // GBK_TO_UNICODE[25966] := 16#CCCB;
   // GBK_TO_UNICODE[25967] := 16#8D9F;
   // GBK_TO_UNICODE[25968] := 16#CCCC;
   // GBK_TO_UNICODE[25969] := 16#70EB;
   // GBK_TO_UNICODE[25970] := 16#CCCD;
   // GBK_TO_UNICODE[25971] := 16#638F;
   // GBK_TO_UNICODE[25972] := 16#CCCE;
   // GBK_TO_UNICODE[25973] := 16#6D9B;
   // GBK_TO_UNICODE[25974] := 16#CCCF;
   // GBK_TO_UNICODE[25975] := 16#6ED4;
   // GBK_TO_UNICODE[25976] := 16#CCD0;
   // GBK_TO_UNICODE[25977] := 16#7EE6;
   // GBK_TO_UNICODE[25978] := 16#CCD1;
   // GBK_TO_UNICODE[25979] := 16#8404;
   // GBK_TO_UNICODE[25980] := 16#CCD2;
   // GBK_TO_UNICODE[25981] := 16#6843;
   // GBK_TO_UNICODE[25982] := 16#CCD3;
   // GBK_TO_UNICODE[25983] := 16#9003;
   // GBK_TO_UNICODE[25984] := 16#CCD4;
   // GBK_TO_UNICODE[25985] := 16#6DD8;
   // GBK_TO_UNICODE[25986] := 16#CCD5;
   // GBK_TO_UNICODE[25987] := 16#9676;
   // GBK_TO_UNICODE[25988] := 16#CCD6;
   // GBK_TO_UNICODE[25989] := 16#8BA8;
   // GBK_TO_UNICODE[25990] := 16#CCD7;
   // GBK_TO_UNICODE[25991] := 16#5957;
   // GBK_TO_UNICODE[25992] := 16#CCD8;
   // GBK_TO_UNICODE[25993] := 16#7279;
   // GBK_TO_UNICODE[25994] := 16#CCD9;
   // GBK_TO_UNICODE[25995] := 16#85E4;
   // GBK_TO_UNICODE[25996] := 16#CCDA;
   // GBK_TO_UNICODE[25997] := 16#817E;
   // GBK_TO_UNICODE[25998] := 16#CCDB;
   // GBK_TO_UNICODE[25999] := 16#75BC;
   // GBK_TO_UNICODE[26000] := 16#CCDC;
   // GBK_TO_UNICODE[26001] := 16#8A8A;
   // GBK_TO_UNICODE[26002] := 16#CCDD;
   // GBK_TO_UNICODE[26003] := 16#68AF;
   // GBK_TO_UNICODE[26004] := 16#CCDE;
   // GBK_TO_UNICODE[26005] := 16#5254;
   // GBK_TO_UNICODE[26006] := 16#CCDF;
   // GBK_TO_UNICODE[26007] := 16#8E22;
   // GBK_TO_UNICODE[26008] := 16#CCE0;
   // GBK_TO_UNICODE[26009] := 16#9511;
   // GBK_TO_UNICODE[26010] := 16#CCE1;
   // GBK_TO_UNICODE[26011] := 16#63D0;
   // GBK_TO_UNICODE[26012] := 16#CCE2;
   // GBK_TO_UNICODE[26013] := 16#9898;
   // GBK_TO_UNICODE[26014] := 16#CCE3;
   // GBK_TO_UNICODE[26015] := 16#8E44;
   // GBK_TO_UNICODE[26016] := 16#CCE4;
   // GBK_TO_UNICODE[26017] := 16#557C;
   // GBK_TO_UNICODE[26018] := 16#CCE5;
   // GBK_TO_UNICODE[26019] := 16#4F53;
   // GBK_TO_UNICODE[26020] := 16#CCE6;
   // GBK_TO_UNICODE[26021] := 16#66FF;
   // GBK_TO_UNICODE[26022] := 16#CCE7;
   // GBK_TO_UNICODE[26023] := 16#568F;
   // GBK_TO_UNICODE[26024] := 16#CCE8;
   // GBK_TO_UNICODE[26025] := 16#60D5;
   // GBK_TO_UNICODE[26026] := 16#CCE9;
   // GBK_TO_UNICODE[26027] := 16#6D95;
   // GBK_TO_UNICODE[26028] := 16#CCEA;
   // GBK_TO_UNICODE[26029] := 16#5243;
   // GBK_TO_UNICODE[26030] := 16#CCEB;
   // GBK_TO_UNICODE[26031] := 16#5C49;
   // GBK_TO_UNICODE[26032] := 16#CCEC;
   // GBK_TO_UNICODE[26033] := 16#5929;
   // GBK_TO_UNICODE[26034] := 16#CCED;
   // GBK_TO_UNICODE[26035] := 16#6DFB;
   // GBK_TO_UNICODE[26036] := 16#CCEE;
   // GBK_TO_UNICODE[26037] := 16#586B;
   // GBK_TO_UNICODE[26038] := 16#CCEF;
   // GBK_TO_UNICODE[26039] := 16#7530;
   // GBK_TO_UNICODE[26040] := 16#CCF0;
   // GBK_TO_UNICODE[26041] := 16#751C;
   // GBK_TO_UNICODE[26042] := 16#CCF1;
   // GBK_TO_UNICODE[26043] := 16#606C;
   // GBK_TO_UNICODE[26044] := 16#CCF2;
   // GBK_TO_UNICODE[26045] := 16#8214;
   // GBK_TO_UNICODE[26046] := 16#CCF3;
   // GBK_TO_UNICODE[26047] := 16#8146;
   // GBK_TO_UNICODE[26048] := 16#CCF4;
   // GBK_TO_UNICODE[26049] := 16#6311;
   // GBK_TO_UNICODE[26050] := 16#CCF5;
   // GBK_TO_UNICODE[26051] := 16#6761;
   // GBK_TO_UNICODE[26052] := 16#CCF6;
   // GBK_TO_UNICODE[26053] := 16#8FE2;
   // GBK_TO_UNICODE[26054] := 16#CCF7;
   // GBK_TO_UNICODE[26055] := 16#773A;
   // GBK_TO_UNICODE[26056] := 16#CCF8;
   // GBK_TO_UNICODE[26057] := 16#8DF3;
   // GBK_TO_UNICODE[26058] := 16#CCF9;
   // GBK_TO_UNICODE[26059] := 16#8D34;
   // GBK_TO_UNICODE[26060] := 16#CCFA;
   // GBK_TO_UNICODE[26061] := 16#94C1;
   // GBK_TO_UNICODE[26062] := 16#CCFB;
   // GBK_TO_UNICODE[26063] := 16#5E16;
   // GBK_TO_UNICODE[26064] := 16#CCFC;
   // GBK_TO_UNICODE[26065] := 16#5385;
   // GBK_TO_UNICODE[26066] := 16#CCFD;
   // GBK_TO_UNICODE[26067] := 16#542C;
   // GBK_TO_UNICODE[26068] := 16#CCFE;
   // GBK_TO_UNICODE[26069] := 16#70C3;
   // GBK_TO_UNICODE[26070] := 16#CD40;
   // GBK_TO_UNICODE[26071] := 16#866D;
   // GBK_TO_UNICODE[26072] := 16#CD41;
   // GBK_TO_UNICODE[26073] := 16#866F;
   // GBK_TO_UNICODE[26074] := 16#CD42;
   // GBK_TO_UNICODE[26075] := 16#8670;
   // GBK_TO_UNICODE[26076] := 16#CD43;
   // GBK_TO_UNICODE[26077] := 16#8672;
   // GBK_TO_UNICODE[26078] := 16#CD44;
   // GBK_TO_UNICODE[26079] := 16#8673;
   // GBK_TO_UNICODE[26080] := 16#CD45;
   // GBK_TO_UNICODE[26081] := 16#8674;
   // GBK_TO_UNICODE[26082] := 16#CD46;
   // GBK_TO_UNICODE[26083] := 16#8675;
   // GBK_TO_UNICODE[26084] := 16#CD47;
   // GBK_TO_UNICODE[26085] := 16#8676;
   // GBK_TO_UNICODE[26086] := 16#CD48;
   // GBK_TO_UNICODE[26087] := 16#8677;
   // GBK_TO_UNICODE[26088] := 16#CD49;
   // GBK_TO_UNICODE[26089] := 16#8678;
   // GBK_TO_UNICODE[26090] := 16#CD4A;
   // GBK_TO_UNICODE[26091] := 16#8683;
   // GBK_TO_UNICODE[26092] := 16#CD4B;
   // GBK_TO_UNICODE[26093] := 16#8684;
   // GBK_TO_UNICODE[26094] := 16#CD4C;
   // GBK_TO_UNICODE[26095] := 16#8685;
   // GBK_TO_UNICODE[26096] := 16#CD4D;
   // GBK_TO_UNICODE[26097] := 16#8686;
   // GBK_TO_UNICODE[26098] := 16#CD4E;
   // GBK_TO_UNICODE[26099] := 16#8687;
   // GBK_TO_UNICODE[26100] := 16#CD4F;
   // GBK_TO_UNICODE[26101] := 16#8688;
   // GBK_TO_UNICODE[26102] := 16#CD50;
   // GBK_TO_UNICODE[26103] := 16#8689;
   // GBK_TO_UNICODE[26104] := 16#CD51;
   // GBK_TO_UNICODE[26105] := 16#868E;
   // GBK_TO_UNICODE[26106] := 16#CD52;
   // GBK_TO_UNICODE[26107] := 16#868F;
   // GBK_TO_UNICODE[26108] := 16#CD53;
   // GBK_TO_UNICODE[26109] := 16#8690;
   // GBK_TO_UNICODE[26110] := 16#CD54;
   // GBK_TO_UNICODE[26111] := 16#8691;
   // GBK_TO_UNICODE[26112] := 16#CD55;
   // GBK_TO_UNICODE[26113] := 16#8692;
   // GBK_TO_UNICODE[26114] := 16#CD56;
   // GBK_TO_UNICODE[26115] := 16#8694;
   // GBK_TO_UNICODE[26116] := 16#CD57;
   // GBK_TO_UNICODE[26117] := 16#8696;
   // GBK_TO_UNICODE[26118] := 16#CD58;
   // GBK_TO_UNICODE[26119] := 16#8697;
   // GBK_TO_UNICODE[26120] := 16#CD59;
   // GBK_TO_UNICODE[26121] := 16#8698;
   // GBK_TO_UNICODE[26122] := 16#CD5A;
   // GBK_TO_UNICODE[26123] := 16#8699;
   // GBK_TO_UNICODE[26124] := 16#CD5B;
   // GBK_TO_UNICODE[26125] := 16#869A;
   // GBK_TO_UNICODE[26126] := 16#CD5C;
   // GBK_TO_UNICODE[26127] := 16#869B;
   // GBK_TO_UNICODE[26128] := 16#CD5D;
   // GBK_TO_UNICODE[26129] := 16#869E;
   // GBK_TO_UNICODE[26130] := 16#CD5E;
   // GBK_TO_UNICODE[26131] := 16#869F;
   // GBK_TO_UNICODE[26132] := 16#CD5F;
   // GBK_TO_UNICODE[26133] := 16#86A0;
   // GBK_TO_UNICODE[26134] := 16#CD60;
   // GBK_TO_UNICODE[26135] := 16#86A1;
   // GBK_TO_UNICODE[26136] := 16#CD61;
   // GBK_TO_UNICODE[26137] := 16#86A2;
   // GBK_TO_UNICODE[26138] := 16#CD62;
   // GBK_TO_UNICODE[26139] := 16#86A5;
   // GBK_TO_UNICODE[26140] := 16#CD63;
   // GBK_TO_UNICODE[26141] := 16#86A6;
   // GBK_TO_UNICODE[26142] := 16#CD64;
   // GBK_TO_UNICODE[26143] := 16#86AB;
   // GBK_TO_UNICODE[26144] := 16#CD65;
   // GBK_TO_UNICODE[26145] := 16#86AD;
   // GBK_TO_UNICODE[26146] := 16#CD66;
   // GBK_TO_UNICODE[26147] := 16#86AE;
   // GBK_TO_UNICODE[26148] := 16#CD67;
   // GBK_TO_UNICODE[26149] := 16#86B2;
   // GBK_TO_UNICODE[26150] := 16#CD68;
   // GBK_TO_UNICODE[26151] := 16#86B3;
   // GBK_TO_UNICODE[26152] := 16#CD69;
   // GBK_TO_UNICODE[26153] := 16#86B7;
   // GBK_TO_UNICODE[26154] := 16#CD6A;
   // GBK_TO_UNICODE[26155] := 16#86B8;
   // GBK_TO_UNICODE[26156] := 16#CD6B;
   // GBK_TO_UNICODE[26157] := 16#86B9;
   // GBK_TO_UNICODE[26158] := 16#CD6C;
   // GBK_TO_UNICODE[26159] := 16#86BB;
   // GBK_TO_UNICODE[26160] := 16#CD6D;
   // GBK_TO_UNICODE[26161] := 16#86BC;
   // GBK_TO_UNICODE[26162] := 16#CD6E;
   // GBK_TO_UNICODE[26163] := 16#86BD;
   // GBK_TO_UNICODE[26164] := 16#CD6F;
   // GBK_TO_UNICODE[26165] := 16#86BE;
   // GBK_TO_UNICODE[26166] := 16#CD70;
   // GBK_TO_UNICODE[26167] := 16#86BF;
   // GBK_TO_UNICODE[26168] := 16#CD71;
   // GBK_TO_UNICODE[26169] := 16#86C1;
   // GBK_TO_UNICODE[26170] := 16#CD72;
   // GBK_TO_UNICODE[26171] := 16#86C2;
   // GBK_TO_UNICODE[26172] := 16#CD73;
   // GBK_TO_UNICODE[26173] := 16#86C3;
   // GBK_TO_UNICODE[26174] := 16#CD74;
   // GBK_TO_UNICODE[26175] := 16#86C5;
   // GBK_TO_UNICODE[26176] := 16#CD75;
   // GBK_TO_UNICODE[26177] := 16#86C8;
   // GBK_TO_UNICODE[26178] := 16#CD76;
   // GBK_TO_UNICODE[26179] := 16#86CC;
   // GBK_TO_UNICODE[26180] := 16#CD77;
   // GBK_TO_UNICODE[26181] := 16#86CD;
   // GBK_TO_UNICODE[26182] := 16#CD78;
   // GBK_TO_UNICODE[26183] := 16#86D2;
   // GBK_TO_UNICODE[26184] := 16#CD79;
   // GBK_TO_UNICODE[26185] := 16#86D3;
   // GBK_TO_UNICODE[26186] := 16#CD7A;
   // GBK_TO_UNICODE[26187] := 16#86D5;
   // GBK_TO_UNICODE[26188] := 16#CD7B;
   // GBK_TO_UNICODE[26189] := 16#86D6;
   // GBK_TO_UNICODE[26190] := 16#CD7C;
   // GBK_TO_UNICODE[26191] := 16#86D7;
   // GBK_TO_UNICODE[26192] := 16#CD7D;
   // GBK_TO_UNICODE[26193] := 16#86DA;
   // GBK_TO_UNICODE[26194] := 16#CD7E;
   // GBK_TO_UNICODE[26195] := 16#86DC;
   // GBK_TO_UNICODE[26196] := 16#CD80;
   // GBK_TO_UNICODE[26197] := 16#86DD;
   // GBK_TO_UNICODE[26198] := 16#CD81;
   // GBK_TO_UNICODE[26199] := 16#86E0;
   // GBK_TO_UNICODE[26200] := 16#CD82;
   // GBK_TO_UNICODE[26201] := 16#86E1;
   // GBK_TO_UNICODE[26202] := 16#CD83;
   // GBK_TO_UNICODE[26203] := 16#86E2;
   // GBK_TO_UNICODE[26204] := 16#CD84;
   // GBK_TO_UNICODE[26205] := 16#86E3;
   // GBK_TO_UNICODE[26206] := 16#CD85;
   // GBK_TO_UNICODE[26207] := 16#86E5;
   // GBK_TO_UNICODE[26208] := 16#CD86;
   // GBK_TO_UNICODE[26209] := 16#86E6;
   // GBK_TO_UNICODE[26210] := 16#CD87;
   // GBK_TO_UNICODE[26211] := 16#86E7;
   // GBK_TO_UNICODE[26212] := 16#CD88;
   // GBK_TO_UNICODE[26213] := 16#86E8;
   // GBK_TO_UNICODE[26214] := 16#CD89;
   // GBK_TO_UNICODE[26215] := 16#86EA;
   // GBK_TO_UNICODE[26216] := 16#CD8A;
   // GBK_TO_UNICODE[26217] := 16#86EB;
   // GBK_TO_UNICODE[26218] := 16#CD8B;
   // GBK_TO_UNICODE[26219] := 16#86EC;
   // GBK_TO_UNICODE[26220] := 16#CD8C;
   // GBK_TO_UNICODE[26221] := 16#86EF;
   // GBK_TO_UNICODE[26222] := 16#CD8D;
   // GBK_TO_UNICODE[26223] := 16#86F5;
   // GBK_TO_UNICODE[26224] := 16#CD8E;
   // GBK_TO_UNICODE[26225] := 16#86F6;
   // GBK_TO_UNICODE[26226] := 16#CD8F;
   // GBK_TO_UNICODE[26227] := 16#86F7;
   // GBK_TO_UNICODE[26228] := 16#CD90;
   // GBK_TO_UNICODE[26229] := 16#86FA;
   // GBK_TO_UNICODE[26230] := 16#CD91;
   // GBK_TO_UNICODE[26231] := 16#86FB;
   // GBK_TO_UNICODE[26232] := 16#CD92;
   // GBK_TO_UNICODE[26233] := 16#86FC;
   // GBK_TO_UNICODE[26234] := 16#CD93;
   // GBK_TO_UNICODE[26235] := 16#86FD;
   // GBK_TO_UNICODE[26236] := 16#CD94;
   // GBK_TO_UNICODE[26237] := 16#86FF;
   // GBK_TO_UNICODE[26238] := 16#CD95;
   // GBK_TO_UNICODE[26239] := 16#8701;
   // GBK_TO_UNICODE[26240] := 16#CD96;
   // GBK_TO_UNICODE[26241] := 16#8704;
   // GBK_TO_UNICODE[26242] := 16#CD97;
   // GBK_TO_UNICODE[26243] := 16#8705;
   // GBK_TO_UNICODE[26244] := 16#CD98;
   // GBK_TO_UNICODE[26245] := 16#8706;
   // GBK_TO_UNICODE[26246] := 16#CD99;
   // GBK_TO_UNICODE[26247] := 16#870B;
   // GBK_TO_UNICODE[26248] := 16#CD9A;
   // GBK_TO_UNICODE[26249] := 16#870C;
   // GBK_TO_UNICODE[26250] := 16#CD9B;
   // GBK_TO_UNICODE[26251] := 16#870E;
   // GBK_TO_UNICODE[26252] := 16#CD9C;
   // GBK_TO_UNICODE[26253] := 16#870F;
   // GBK_TO_UNICODE[26254] := 16#CD9D;
   // GBK_TO_UNICODE[26255] := 16#8710;
   // GBK_TO_UNICODE[26256] := 16#CD9E;
   // GBK_TO_UNICODE[26257] := 16#8711;
   // GBK_TO_UNICODE[26258] := 16#CD9F;
   // GBK_TO_UNICODE[26259] := 16#8714;
   // GBK_TO_UNICODE[26260] := 16#CDA0;
   // GBK_TO_UNICODE[26261] := 16#8716;
   // GBK_TO_UNICODE[26262] := 16#CDA1;
   // GBK_TO_UNICODE[26263] := 16#6C40;
   // GBK_TO_UNICODE[26264] := 16#CDA2;
   // GBK_TO_UNICODE[26265] := 16#5EF7;
   // GBK_TO_UNICODE[26266] := 16#CDA3;
   // GBK_TO_UNICODE[26267] := 16#505C;
   // GBK_TO_UNICODE[26268] := 16#CDA4;
   // GBK_TO_UNICODE[26269] := 16#4EAD;
   // GBK_TO_UNICODE[26270] := 16#CDA5;
   // GBK_TO_UNICODE[26271] := 16#5EAD;
   // GBK_TO_UNICODE[26272] := 16#CDA6;
   // GBK_TO_UNICODE[26273] := 16#633A;
   // GBK_TO_UNICODE[26274] := 16#CDA7;
   // GBK_TO_UNICODE[26275] := 16#8247;
   // GBK_TO_UNICODE[26276] := 16#CDA8;
   // GBK_TO_UNICODE[26277] := 16#901A;
   // GBK_TO_UNICODE[26278] := 16#CDA9;
   // GBK_TO_UNICODE[26279] := 16#6850;
   // GBK_TO_UNICODE[26280] := 16#CDAA;
   // GBK_TO_UNICODE[26281] := 16#916E;
   // GBK_TO_UNICODE[26282] := 16#CDAB;
   // GBK_TO_UNICODE[26283] := 16#77B3;
   // GBK_TO_UNICODE[26284] := 16#CDAC;
   // GBK_TO_UNICODE[26285] := 16#540C;
   // GBK_TO_UNICODE[26286] := 16#CDAD;
   // GBK_TO_UNICODE[26287] := 16#94DC;
   // GBK_TO_UNICODE[26288] := 16#CDAE;
   // GBK_TO_UNICODE[26289] := 16#5F64;
   // GBK_TO_UNICODE[26290] := 16#CDAF;
   // GBK_TO_UNICODE[26291] := 16#7AE5;
   // GBK_TO_UNICODE[26292] := 16#CDB0;
   // GBK_TO_UNICODE[26293] := 16#6876;
   // GBK_TO_UNICODE[26294] := 16#CDB1;
   // GBK_TO_UNICODE[26295] := 16#6345;
   // GBK_TO_UNICODE[26296] := 16#CDB2;
   // GBK_TO_UNICODE[26297] := 16#7B52;
   // GBK_TO_UNICODE[26298] := 16#CDB3;
   // GBK_TO_UNICODE[26299] := 16#7EDF;
   // GBK_TO_UNICODE[26300] := 16#CDB4;
   // GBK_TO_UNICODE[26301] := 16#75DB;
   // GBK_TO_UNICODE[26302] := 16#CDB5;
   // GBK_TO_UNICODE[26303] := 16#5077;
   // GBK_TO_UNICODE[26304] := 16#CDB6;
   // GBK_TO_UNICODE[26305] := 16#6295;
   // GBK_TO_UNICODE[26306] := 16#CDB7;
   // GBK_TO_UNICODE[26307] := 16#5934;
   // GBK_TO_UNICODE[26308] := 16#CDB8;
   // GBK_TO_UNICODE[26309] := 16#900F;
   // GBK_TO_UNICODE[26310] := 16#CDB9;
   // GBK_TO_UNICODE[26311] := 16#51F8;
   // GBK_TO_UNICODE[26312] := 16#CDBA;
   // GBK_TO_UNICODE[26313] := 16#79C3;
   // GBK_TO_UNICODE[26314] := 16#CDBB;
   // GBK_TO_UNICODE[26315] := 16#7A81;
   // GBK_TO_UNICODE[26316] := 16#CDBC;
   // GBK_TO_UNICODE[26317] := 16#56FE;
   // GBK_TO_UNICODE[26318] := 16#CDBD;
   // GBK_TO_UNICODE[26319] := 16#5F92;
   // GBK_TO_UNICODE[26320] := 16#CDBE;
   // GBK_TO_UNICODE[26321] := 16#9014;
   // GBK_TO_UNICODE[26322] := 16#CDBF;
   // GBK_TO_UNICODE[26323] := 16#6D82;
   // GBK_TO_UNICODE[26324] := 16#CDC0;
   // GBK_TO_UNICODE[26325] := 16#5C60;
   // GBK_TO_UNICODE[26326] := 16#CDC1;
   // GBK_TO_UNICODE[26327] := 16#571F;
   // GBK_TO_UNICODE[26328] := 16#CDC2;
   // GBK_TO_UNICODE[26329] := 16#5410;
   // GBK_TO_UNICODE[26330] := 16#CDC3;
   // GBK_TO_UNICODE[26331] := 16#5154;
   // GBK_TO_UNICODE[26332] := 16#CDC4;
   // GBK_TO_UNICODE[26333] := 16#6E4D;
   // GBK_TO_UNICODE[26334] := 16#CDC5;
   // GBK_TO_UNICODE[26335] := 16#56E2;
   // GBK_TO_UNICODE[26336] := 16#CDC6;
   // GBK_TO_UNICODE[26337] := 16#63A8;
   // GBK_TO_UNICODE[26338] := 16#CDC7;
   // GBK_TO_UNICODE[26339] := 16#9893;
   // GBK_TO_UNICODE[26340] := 16#CDC8;
   // GBK_TO_UNICODE[26341] := 16#817F;
   // GBK_TO_UNICODE[26342] := 16#CDC9;
   // GBK_TO_UNICODE[26343] := 16#8715;
   // GBK_TO_UNICODE[26344] := 16#CDCA;
   // GBK_TO_UNICODE[26345] := 16#892A;
   // GBK_TO_UNICODE[26346] := 16#CDCB;
   // GBK_TO_UNICODE[26347] := 16#9000;
   // GBK_TO_UNICODE[26348] := 16#CDCC;
   // GBK_TO_UNICODE[26349] := 16#541E;
   // GBK_TO_UNICODE[26350] := 16#CDCD;
   // GBK_TO_UNICODE[26351] := 16#5C6F;
   // GBK_TO_UNICODE[26352] := 16#CDCE;
   // GBK_TO_UNICODE[26353] := 16#81C0;
   // GBK_TO_UNICODE[26354] := 16#CDCF;
   // GBK_TO_UNICODE[26355] := 16#62D6;
   // GBK_TO_UNICODE[26356] := 16#CDD0;
   // GBK_TO_UNICODE[26357] := 16#6258;
   // GBK_TO_UNICODE[26358] := 16#CDD1;
   // GBK_TO_UNICODE[26359] := 16#8131;
   // GBK_TO_UNICODE[26360] := 16#CDD2;
   // GBK_TO_UNICODE[26361] := 16#9E35;
   // GBK_TO_UNICODE[26362] := 16#CDD3;
   // GBK_TO_UNICODE[26363] := 16#9640;
   // GBK_TO_UNICODE[26364] := 16#CDD4;
   // GBK_TO_UNICODE[26365] := 16#9A6E;
   // GBK_TO_UNICODE[26366] := 16#CDD5;
   // GBK_TO_UNICODE[26367] := 16#9A7C;
   // GBK_TO_UNICODE[26368] := 16#CDD6;
   // GBK_TO_UNICODE[26369] := 16#692D;
   // GBK_TO_UNICODE[26370] := 16#CDD7;
   // GBK_TO_UNICODE[26371] := 16#59A5;
   // GBK_TO_UNICODE[26372] := 16#CDD8;
   // GBK_TO_UNICODE[26373] := 16#62D3;
   // GBK_TO_UNICODE[26374] := 16#CDD9;
   // GBK_TO_UNICODE[26375] := 16#553E;
   // GBK_TO_UNICODE[26376] := 16#CDDA;
   // GBK_TO_UNICODE[26377] := 16#6316;
   // GBK_TO_UNICODE[26378] := 16#CDDB;
   // GBK_TO_UNICODE[26379] := 16#54C7;
   // GBK_TO_UNICODE[26380] := 16#CDDC;
   // GBK_TO_UNICODE[26381] := 16#86D9;
   // GBK_TO_UNICODE[26382] := 16#CDDD;
   // GBK_TO_UNICODE[26383] := 16#6D3C;
   // GBK_TO_UNICODE[26384] := 16#CDDE;
   // GBK_TO_UNICODE[26385] := 16#5A03;
   // GBK_TO_UNICODE[26386] := 16#CDDF;
   // GBK_TO_UNICODE[26387] := 16#74E6;
   // GBK_TO_UNICODE[26388] := 16#CDE0;
   // GBK_TO_UNICODE[26389] := 16#889C;
   // GBK_TO_UNICODE[26390] := 16#CDE1;
   // GBK_TO_UNICODE[26391] := 16#6B6A;
   // GBK_TO_UNICODE[26392] := 16#CDE2;
   // GBK_TO_UNICODE[26393] := 16#5916;
   // GBK_TO_UNICODE[26394] := 16#CDE3;
   // GBK_TO_UNICODE[26395] := 16#8C4C;
   // GBK_TO_UNICODE[26396] := 16#CDE4;
   // GBK_TO_UNICODE[26397] := 16#5F2F;
   // GBK_TO_UNICODE[26398] := 16#CDE5;
   // GBK_TO_UNICODE[26399] := 16#6E7E;
   // GBK_TO_UNICODE[26400] := 16#CDE6;
   // GBK_TO_UNICODE[26401] := 16#73A9;
   // GBK_TO_UNICODE[26402] := 16#CDE7;
   // GBK_TO_UNICODE[26403] := 16#987D;
   // GBK_TO_UNICODE[26404] := 16#CDE8;
   // GBK_TO_UNICODE[26405] := 16#4E38;
   // GBK_TO_UNICODE[26406] := 16#CDE9;
   // GBK_TO_UNICODE[26407] := 16#70F7;
   // GBK_TO_UNICODE[26408] := 16#CDEA;
   // GBK_TO_UNICODE[26409] := 16#5B8C;
   // GBK_TO_UNICODE[26410] := 16#CDEB;
   // GBK_TO_UNICODE[26411] := 16#7897;
   // GBK_TO_UNICODE[26412] := 16#CDEC;
   // GBK_TO_UNICODE[26413] := 16#633D;
   // GBK_TO_UNICODE[26414] := 16#CDED;
   // GBK_TO_UNICODE[26415] := 16#665A;
   // GBK_TO_UNICODE[26416] := 16#CDEE;
   // GBK_TO_UNICODE[26417] := 16#7696;
   // GBK_TO_UNICODE[26418] := 16#CDEF;
   // GBK_TO_UNICODE[26419] := 16#60CB;
   // GBK_TO_UNICODE[26420] := 16#CDF0;
   // GBK_TO_UNICODE[26421] := 16#5B9B;
   // GBK_TO_UNICODE[26422] := 16#CDF1;
   // GBK_TO_UNICODE[26423] := 16#5A49;
   // GBK_TO_UNICODE[26424] := 16#CDF2;
   // GBK_TO_UNICODE[26425] := 16#4E07;
   // GBK_TO_UNICODE[26426] := 16#CDF3;
   // GBK_TO_UNICODE[26427] := 16#8155;
   // GBK_TO_UNICODE[26428] := 16#CDF4;
   // GBK_TO_UNICODE[26429] := 16#6C6A;
   // GBK_TO_UNICODE[26430] := 16#CDF5;
   // GBK_TO_UNICODE[26431] := 16#738B;
   // GBK_TO_UNICODE[26432] := 16#CDF6;
   // GBK_TO_UNICODE[26433] := 16#4EA1;
   // GBK_TO_UNICODE[26434] := 16#CDF7;
   // GBK_TO_UNICODE[26435] := 16#6789;
   // GBK_TO_UNICODE[26436] := 16#CDF8;
   // GBK_TO_UNICODE[26437] := 16#7F51;
   // GBK_TO_UNICODE[26438] := 16#CDF9;
   // GBK_TO_UNICODE[26439] := 16#5F80;
   // GBK_TO_UNICODE[26440] := 16#CDFA;
   // GBK_TO_UNICODE[26441] := 16#65FA;
   // GBK_TO_UNICODE[26442] := 16#CDFB;
   // GBK_TO_UNICODE[26443] := 16#671B;
   // GBK_TO_UNICODE[26444] := 16#CDFC;
   // GBK_TO_UNICODE[26445] := 16#5FD8;
   // GBK_TO_UNICODE[26446] := 16#CDFD;
   // GBK_TO_UNICODE[26447] := 16#5984;
   // GBK_TO_UNICODE[26448] := 16#CDFE;
   // GBK_TO_UNICODE[26449] := 16#5A01;
   // GBK_TO_UNICODE[26450] := 16#CE40;
   // GBK_TO_UNICODE[26451] := 16#8719;
   // GBK_TO_UNICODE[26452] := 16#CE41;
   // GBK_TO_UNICODE[26453] := 16#871B;
   // GBK_TO_UNICODE[26454] := 16#CE42;
   // GBK_TO_UNICODE[26455] := 16#871D;
   // GBK_TO_UNICODE[26456] := 16#CE43;
   // GBK_TO_UNICODE[26457] := 16#871F;
   // GBK_TO_UNICODE[26458] := 16#CE44;
   // GBK_TO_UNICODE[26459] := 16#8720;
   // GBK_TO_UNICODE[26460] := 16#CE45;
   // GBK_TO_UNICODE[26461] := 16#8724;
   // GBK_TO_UNICODE[26462] := 16#CE46;
   // GBK_TO_UNICODE[26463] := 16#8726;
   // GBK_TO_UNICODE[26464] := 16#CE47;
   // GBK_TO_UNICODE[26465] := 16#8727;
   // GBK_TO_UNICODE[26466] := 16#CE48;
   // GBK_TO_UNICODE[26467] := 16#8728;
   // GBK_TO_UNICODE[26468] := 16#CE49;
   // GBK_TO_UNICODE[26469] := 16#872A;
   // GBK_TO_UNICODE[26470] := 16#CE4A;
   // GBK_TO_UNICODE[26471] := 16#872B;
   // GBK_TO_UNICODE[26472] := 16#CE4B;
   // GBK_TO_UNICODE[26473] := 16#872C;
   // GBK_TO_UNICODE[26474] := 16#CE4C;
   // GBK_TO_UNICODE[26475] := 16#872D;
   // GBK_TO_UNICODE[26476] := 16#CE4D;
   // GBK_TO_UNICODE[26477] := 16#872F;
   // GBK_TO_UNICODE[26478] := 16#CE4E;
   // GBK_TO_UNICODE[26479] := 16#8730;
   // GBK_TO_UNICODE[26480] := 16#CE4F;
   // GBK_TO_UNICODE[26481] := 16#8732;
   // GBK_TO_UNICODE[26482] := 16#CE50;
   // GBK_TO_UNICODE[26483] := 16#8733;
   // GBK_TO_UNICODE[26484] := 16#CE51;
   // GBK_TO_UNICODE[26485] := 16#8735;
   // GBK_TO_UNICODE[26486] := 16#CE52;
   // GBK_TO_UNICODE[26487] := 16#8736;
   // GBK_TO_UNICODE[26488] := 16#CE53;
   // GBK_TO_UNICODE[26489] := 16#8738;
   // GBK_TO_UNICODE[26490] := 16#CE54;
   // GBK_TO_UNICODE[26491] := 16#8739;
   // GBK_TO_UNICODE[26492] := 16#CE55;
   // GBK_TO_UNICODE[26493] := 16#873A;
   // GBK_TO_UNICODE[26494] := 16#CE56;
   // GBK_TO_UNICODE[26495] := 16#873C;
   // GBK_TO_UNICODE[26496] := 16#CE57;
   // GBK_TO_UNICODE[26497] := 16#873D;
   // GBK_TO_UNICODE[26498] := 16#CE58;
   // GBK_TO_UNICODE[26499] := 16#8740;
   // GBK_TO_UNICODE[26500] := 16#CE59;
   // GBK_TO_UNICODE[26501] := 16#8741;
   // GBK_TO_UNICODE[26502] := 16#CE5A;
   // GBK_TO_UNICODE[26503] := 16#8742;
   // GBK_TO_UNICODE[26504] := 16#CE5B;
   // GBK_TO_UNICODE[26505] := 16#8743;
   // GBK_TO_UNICODE[26506] := 16#CE5C;
   // GBK_TO_UNICODE[26507] := 16#8744;
   // GBK_TO_UNICODE[26508] := 16#CE5D;
   // GBK_TO_UNICODE[26509] := 16#8745;
   // GBK_TO_UNICODE[26510] := 16#CE5E;
   // GBK_TO_UNICODE[26511] := 16#8746;
   // GBK_TO_UNICODE[26512] := 16#CE5F;
   // GBK_TO_UNICODE[26513] := 16#874A;
   // GBK_TO_UNICODE[26514] := 16#CE60;
   // GBK_TO_UNICODE[26515] := 16#874B;
   // GBK_TO_UNICODE[26516] := 16#CE61;
   // GBK_TO_UNICODE[26517] := 16#874D;
   // GBK_TO_UNICODE[26518] := 16#CE62;
   // GBK_TO_UNICODE[26519] := 16#874F;
   // GBK_TO_UNICODE[26520] := 16#CE63;
   // GBK_TO_UNICODE[26521] := 16#8750;
   // GBK_TO_UNICODE[26522] := 16#CE64;
   // GBK_TO_UNICODE[26523] := 16#8751;
   // GBK_TO_UNICODE[26524] := 16#CE65;
   // GBK_TO_UNICODE[26525] := 16#8752;
   // GBK_TO_UNICODE[26526] := 16#CE66;
   // GBK_TO_UNICODE[26527] := 16#8754;
   // GBK_TO_UNICODE[26528] := 16#CE67;
   // GBK_TO_UNICODE[26529] := 16#8755;
   // GBK_TO_UNICODE[26530] := 16#CE68;
   // GBK_TO_UNICODE[26531] := 16#8756;
   // GBK_TO_UNICODE[26532] := 16#CE69;
   // GBK_TO_UNICODE[26533] := 16#8758;
   // GBK_TO_UNICODE[26534] := 16#CE6A;
   // GBK_TO_UNICODE[26535] := 16#875A;
   // GBK_TO_UNICODE[26536] := 16#CE6B;
   // GBK_TO_UNICODE[26537] := 16#875B;
   // GBK_TO_UNICODE[26538] := 16#CE6C;
   // GBK_TO_UNICODE[26539] := 16#875C;
   // GBK_TO_UNICODE[26540] := 16#CE6D;
   // GBK_TO_UNICODE[26541] := 16#875D;
   // GBK_TO_UNICODE[26542] := 16#CE6E;
   // GBK_TO_UNICODE[26543] := 16#875E;
   // GBK_TO_UNICODE[26544] := 16#CE6F;
   // GBK_TO_UNICODE[26545] := 16#875F;
   // GBK_TO_UNICODE[26546] := 16#CE70;
   // GBK_TO_UNICODE[26547] := 16#8761;
   // GBK_TO_UNICODE[26548] := 16#CE71;
   // GBK_TO_UNICODE[26549] := 16#8762;
   // GBK_TO_UNICODE[26550] := 16#CE72;
   // GBK_TO_UNICODE[26551] := 16#8766;
   // GBK_TO_UNICODE[26552] := 16#CE73;
   // GBK_TO_UNICODE[26553] := 16#8767;
   // GBK_TO_UNICODE[26554] := 16#CE74;
   // GBK_TO_UNICODE[26555] := 16#8768;
   // GBK_TO_UNICODE[26556] := 16#CE75;
   // GBK_TO_UNICODE[26557] := 16#8769;
   // GBK_TO_UNICODE[26558] := 16#CE76;
   // GBK_TO_UNICODE[26559] := 16#876A;
   // GBK_TO_UNICODE[26560] := 16#CE77;
   // GBK_TO_UNICODE[26561] := 16#876B;
   // GBK_TO_UNICODE[26562] := 16#CE78;
   // GBK_TO_UNICODE[26563] := 16#876C;
   // GBK_TO_UNICODE[26564] := 16#CE79;
   // GBK_TO_UNICODE[26565] := 16#876D;
   // GBK_TO_UNICODE[26566] := 16#CE7A;
   // GBK_TO_UNICODE[26567] := 16#876F;
   // GBK_TO_UNICODE[26568] := 16#CE7B;
   // GBK_TO_UNICODE[26569] := 16#8771;
   // GBK_TO_UNICODE[26570] := 16#CE7C;
   // GBK_TO_UNICODE[26571] := 16#8772;
   // GBK_TO_UNICODE[26572] := 16#CE7D;
   // GBK_TO_UNICODE[26573] := 16#8773;
   // GBK_TO_UNICODE[26574] := 16#CE7E;
   // GBK_TO_UNICODE[26575] := 16#8775;
   // GBK_TO_UNICODE[26576] := 16#CE80;
   // GBK_TO_UNICODE[26577] := 16#8777;
   // GBK_TO_UNICODE[26578] := 16#CE81;
   // GBK_TO_UNICODE[26579] := 16#8778;
   // GBK_TO_UNICODE[26580] := 16#CE82;
   // GBK_TO_UNICODE[26581] := 16#8779;
   // GBK_TO_UNICODE[26582] := 16#CE83;
   // GBK_TO_UNICODE[26583] := 16#877A;
   // GBK_TO_UNICODE[26584] := 16#CE84;
   // GBK_TO_UNICODE[26585] := 16#877F;
   // GBK_TO_UNICODE[26586] := 16#CE85;
   // GBK_TO_UNICODE[26587] := 16#8780;
   // GBK_TO_UNICODE[26588] := 16#CE86;
   // GBK_TO_UNICODE[26589] := 16#8781;
   // GBK_TO_UNICODE[26590] := 16#CE87;
   // GBK_TO_UNICODE[26591] := 16#8784;
   // GBK_TO_UNICODE[26592] := 16#CE88;
   // GBK_TO_UNICODE[26593] := 16#8786;
   // GBK_TO_UNICODE[26594] := 16#CE89;
   // GBK_TO_UNICODE[26595] := 16#8787;
   // GBK_TO_UNICODE[26596] := 16#CE8A;
   // GBK_TO_UNICODE[26597] := 16#8789;
   // GBK_TO_UNICODE[26598] := 16#CE8B;
   // GBK_TO_UNICODE[26599] := 16#878A;
   // GBK_TO_UNICODE[26600] := 16#CE8C;
   // GBK_TO_UNICODE[26601] := 16#878C;
   // GBK_TO_UNICODE[26602] := 16#CE8D;
   // GBK_TO_UNICODE[26603] := 16#878E;
   // GBK_TO_UNICODE[26604] := 16#CE8E;
   // GBK_TO_UNICODE[26605] := 16#878F;
   // GBK_TO_UNICODE[26606] := 16#CE8F;
   // GBK_TO_UNICODE[26607] := 16#8790;
   // GBK_TO_UNICODE[26608] := 16#CE90;
   // GBK_TO_UNICODE[26609] := 16#8791;
   // GBK_TO_UNICODE[26610] := 16#CE91;
   // GBK_TO_UNICODE[26611] := 16#8792;
   // GBK_TO_UNICODE[26612] := 16#CE92;
   // GBK_TO_UNICODE[26613] := 16#8794;
   // GBK_TO_UNICODE[26614] := 16#CE93;
   // GBK_TO_UNICODE[26615] := 16#8795;
   // GBK_TO_UNICODE[26616] := 16#CE94;
   // GBK_TO_UNICODE[26617] := 16#8796;
   // GBK_TO_UNICODE[26618] := 16#CE95;
   // GBK_TO_UNICODE[26619] := 16#8798;
   // GBK_TO_UNICODE[26620] := 16#CE96;
   // GBK_TO_UNICODE[26621] := 16#8799;
   // GBK_TO_UNICODE[26622] := 16#CE97;
   // GBK_TO_UNICODE[26623] := 16#879A;
   // GBK_TO_UNICODE[26624] := 16#CE98;
   // GBK_TO_UNICODE[26625] := 16#879B;
   // GBK_TO_UNICODE[26626] := 16#CE99;
   // GBK_TO_UNICODE[26627] := 16#879C;
   // GBK_TO_UNICODE[26628] := 16#CE9A;
   // GBK_TO_UNICODE[26629] := 16#879D;
   // GBK_TO_UNICODE[26630] := 16#CE9B;
   // GBK_TO_UNICODE[26631] := 16#879E;
   // GBK_TO_UNICODE[26632] := 16#CE9C;
   // GBK_TO_UNICODE[26633] := 16#87A0;
   // GBK_TO_UNICODE[26634] := 16#CE9D;
   // GBK_TO_UNICODE[26635] := 16#87A1;
   // GBK_TO_UNICODE[26636] := 16#CE9E;
   // GBK_TO_UNICODE[26637] := 16#87A2;
   // GBK_TO_UNICODE[26638] := 16#CE9F;
   // GBK_TO_UNICODE[26639] := 16#87A3;
   // GBK_TO_UNICODE[26640] := 16#CEA0;
   // GBK_TO_UNICODE[26641] := 16#87A4;
   // GBK_TO_UNICODE[26642] := 16#CEA1;
   // GBK_TO_UNICODE[26643] := 16#5DCD;
   // GBK_TO_UNICODE[26644] := 16#CEA2;
   // GBK_TO_UNICODE[26645] := 16#5FAE;
   // GBK_TO_UNICODE[26646] := 16#CEA3;
   // GBK_TO_UNICODE[26647] := 16#5371;
   // GBK_TO_UNICODE[26648] := 16#CEA4;
   // GBK_TO_UNICODE[26649] := 16#97E6;
   // GBK_TO_UNICODE[26650] := 16#CEA5;
   // GBK_TO_UNICODE[26651] := 16#8FDD;
   // GBK_TO_UNICODE[26652] := 16#CEA6;
   // GBK_TO_UNICODE[26653] := 16#6845;
   // GBK_TO_UNICODE[26654] := 16#CEA7;
   // GBK_TO_UNICODE[26655] := 16#56F4;
   // GBK_TO_UNICODE[26656] := 16#CEA8;
   // GBK_TO_UNICODE[26657] := 16#552F;
   // GBK_TO_UNICODE[26658] := 16#CEA9;
   // GBK_TO_UNICODE[26659] := 16#60DF;
   // GBK_TO_UNICODE[26660] := 16#CEAA;
   // GBK_TO_UNICODE[26661] := 16#4E3A;
   // GBK_TO_UNICODE[26662] := 16#CEAB;
   // GBK_TO_UNICODE[26663] := 16#6F4D;
   // GBK_TO_UNICODE[26664] := 16#CEAC;
   // GBK_TO_UNICODE[26665] := 16#7EF4;
   // GBK_TO_UNICODE[26666] := 16#CEAD;
   // GBK_TO_UNICODE[26667] := 16#82C7;
   // GBK_TO_UNICODE[26668] := 16#CEAE;
   // GBK_TO_UNICODE[26669] := 16#840E;
   // GBK_TO_UNICODE[26670] := 16#CEAF;
   // GBK_TO_UNICODE[26671] := 16#59D4;
   // GBK_TO_UNICODE[26672] := 16#CEB0;
   // GBK_TO_UNICODE[26673] := 16#4F1F;
   // GBK_TO_UNICODE[26674] := 16#CEB1;
   // GBK_TO_UNICODE[26675] := 16#4F2A;
   // GBK_TO_UNICODE[26676] := 16#CEB2;
   // GBK_TO_UNICODE[26677] := 16#5C3E;
   // GBK_TO_UNICODE[26678] := 16#CEB3;
   // GBK_TO_UNICODE[26679] := 16#7EAC;
   // GBK_TO_UNICODE[26680] := 16#CEB4;
   // GBK_TO_UNICODE[26681] := 16#672A;
   // GBK_TO_UNICODE[26682] := 16#CEB5;
   // GBK_TO_UNICODE[26683] := 16#851A;
   // GBK_TO_UNICODE[26684] := 16#CEB6;
   // GBK_TO_UNICODE[26685] := 16#5473;
   // GBK_TO_UNICODE[26686] := 16#CEB7;
   // GBK_TO_UNICODE[26687] := 16#754F;
   // GBK_TO_UNICODE[26688] := 16#CEB8;
   // GBK_TO_UNICODE[26689] := 16#80C3;
   // GBK_TO_UNICODE[26690] := 16#CEB9;
   // GBK_TO_UNICODE[26691] := 16#5582;
   // GBK_TO_UNICODE[26692] := 16#CEBA;
   // GBK_TO_UNICODE[26693] := 16#9B4F;
   // GBK_TO_UNICODE[26694] := 16#CEBB;
   // GBK_TO_UNICODE[26695] := 16#4F4D;
   // GBK_TO_UNICODE[26696] := 16#CEBC;
   // GBK_TO_UNICODE[26697] := 16#6E2D;
   // GBK_TO_UNICODE[26698] := 16#CEBD;
   // GBK_TO_UNICODE[26699] := 16#8C13;
   // GBK_TO_UNICODE[26700] := 16#CEBE;
   // GBK_TO_UNICODE[26701] := 16#5C09;
   // GBK_TO_UNICODE[26702] := 16#CEBF;
   // GBK_TO_UNICODE[26703] := 16#6170;
   // GBK_TO_UNICODE[26704] := 16#CEC0;
   // GBK_TO_UNICODE[26705] := 16#536B;
   // GBK_TO_UNICODE[26706] := 16#CEC1;
   // GBK_TO_UNICODE[26707] := 16#761F;
   // GBK_TO_UNICODE[26708] := 16#CEC2;
   // GBK_TO_UNICODE[26709] := 16#6E29;
   // GBK_TO_UNICODE[26710] := 16#CEC3;
   // GBK_TO_UNICODE[26711] := 16#868A;
   // GBK_TO_UNICODE[26712] := 16#CEC4;
   // GBK_TO_UNICODE[26713] := 16#6587;
   // GBK_TO_UNICODE[26714] := 16#CEC5;
   // GBK_TO_UNICODE[26715] := 16#95FB;
   // GBK_TO_UNICODE[26716] := 16#CEC6;
   // GBK_TO_UNICODE[26717] := 16#7EB9;
   // GBK_TO_UNICODE[26718] := 16#CEC7;
   // GBK_TO_UNICODE[26719] := 16#543B;
   // GBK_TO_UNICODE[26720] := 16#CEC8;
   // GBK_TO_UNICODE[26721] := 16#7A33;
   // GBK_TO_UNICODE[26722] := 16#CEC9;
   // GBK_TO_UNICODE[26723] := 16#7D0A;
   // GBK_TO_UNICODE[26724] := 16#CECA;
   // GBK_TO_UNICODE[26725] := 16#95EE;
   // GBK_TO_UNICODE[26726] := 16#CECB;
   // GBK_TO_UNICODE[26727] := 16#55E1;
   // GBK_TO_UNICODE[26728] := 16#CECC;
   // GBK_TO_UNICODE[26729] := 16#7FC1;
   // GBK_TO_UNICODE[26730] := 16#CECD;
   // GBK_TO_UNICODE[26731] := 16#74EE;
   // GBK_TO_UNICODE[26732] := 16#CECE;
   // GBK_TO_UNICODE[26733] := 16#631D;
   // GBK_TO_UNICODE[26734] := 16#CECF;
   // GBK_TO_UNICODE[26735] := 16#8717;
   // GBK_TO_UNICODE[26736] := 16#CED0;
   // GBK_TO_UNICODE[26737] := 16#6DA1;
   // GBK_TO_UNICODE[26738] := 16#CED1;
   // GBK_TO_UNICODE[26739] := 16#7A9D;
   // GBK_TO_UNICODE[26740] := 16#CED2;
   // GBK_TO_UNICODE[26741] := 16#6211;
   // GBK_TO_UNICODE[26742] := 16#CED3;
   // GBK_TO_UNICODE[26743] := 16#65A1;
   // GBK_TO_UNICODE[26744] := 16#CED4;
   // GBK_TO_UNICODE[26745] := 16#5367;
   // GBK_TO_UNICODE[26746] := 16#CED5;
   // GBK_TO_UNICODE[26747] := 16#63E1;
   // GBK_TO_UNICODE[26748] := 16#CED6;
   // GBK_TO_UNICODE[26749] := 16#6C83;
   // GBK_TO_UNICODE[26750] := 16#CED7;
   // GBK_TO_UNICODE[26751] := 16#5DEB;
   // GBK_TO_UNICODE[26752] := 16#CED8;
   // GBK_TO_UNICODE[26753] := 16#545C;
   // GBK_TO_UNICODE[26754] := 16#CED9;
   // GBK_TO_UNICODE[26755] := 16#94A8;
   // GBK_TO_UNICODE[26756] := 16#CEDA;
   // GBK_TO_UNICODE[26757] := 16#4E4C;
   // GBK_TO_UNICODE[26758] := 16#CEDB;
   // GBK_TO_UNICODE[26759] := 16#6C61;
   // GBK_TO_UNICODE[26760] := 16#CEDC;
   // GBK_TO_UNICODE[26761] := 16#8BEC;
   // GBK_TO_UNICODE[26762] := 16#CEDD;
   // GBK_TO_UNICODE[26763] := 16#5C4B;
   // GBK_TO_UNICODE[26764] := 16#CEDE;
   // GBK_TO_UNICODE[26765] := 16#65E0;
   // GBK_TO_UNICODE[26766] := 16#CEDF;
   // GBK_TO_UNICODE[26767] := 16#829C;
   // GBK_TO_UNICODE[26768] := 16#CEE0;
   // GBK_TO_UNICODE[26769] := 16#68A7;
   // GBK_TO_UNICODE[26770] := 16#CEE1;
   // GBK_TO_UNICODE[26771] := 16#543E;
   // GBK_TO_UNICODE[26772] := 16#CEE2;
   // GBK_TO_UNICODE[26773] := 16#5434;
   // GBK_TO_UNICODE[26774] := 16#CEE3;
   // GBK_TO_UNICODE[26775] := 16#6BCB;
   // GBK_TO_UNICODE[26776] := 16#CEE4;
   // GBK_TO_UNICODE[26777] := 16#6B66;
   // GBK_TO_UNICODE[26778] := 16#CEE5;
   // GBK_TO_UNICODE[26779] := 16#4E94;
   // GBK_TO_UNICODE[26780] := 16#CEE6;
   // GBK_TO_UNICODE[26781] := 16#6342;
   // GBK_TO_UNICODE[26782] := 16#CEE7;
   // GBK_TO_UNICODE[26783] := 16#5348;
   // GBK_TO_UNICODE[26784] := 16#CEE8;
   // GBK_TO_UNICODE[26785] := 16#821E;
   // GBK_TO_UNICODE[26786] := 16#CEE9;
   // GBK_TO_UNICODE[26787] := 16#4F0D;
   // GBK_TO_UNICODE[26788] := 16#CEEA;
   // GBK_TO_UNICODE[26789] := 16#4FAE;
   // GBK_TO_UNICODE[26790] := 16#CEEB;
   // GBK_TO_UNICODE[26791] := 16#575E;
   // GBK_TO_UNICODE[26792] := 16#CEEC;
   // GBK_TO_UNICODE[26793] := 16#620A;
   // GBK_TO_UNICODE[26794] := 16#CEED;
   // GBK_TO_UNICODE[26795] := 16#96FE;
   // GBK_TO_UNICODE[26796] := 16#CEEE;
   // GBK_TO_UNICODE[26797] := 16#6664;
   // GBK_TO_UNICODE[26798] := 16#CEEF;
   // GBK_TO_UNICODE[26799] := 16#7269;
   // GBK_TO_UNICODE[26800] := 16#CEF0;
   // GBK_TO_UNICODE[26801] := 16#52FF;
   // GBK_TO_UNICODE[26802] := 16#CEF1;
   // GBK_TO_UNICODE[26803] := 16#52A1;
   // GBK_TO_UNICODE[26804] := 16#CEF2;
   // GBK_TO_UNICODE[26805] := 16#609F;
   // GBK_TO_UNICODE[26806] := 16#CEF3;
   // GBK_TO_UNICODE[26807] := 16#8BEF;
   // GBK_TO_UNICODE[26808] := 16#CEF4;
   // GBK_TO_UNICODE[26809] := 16#6614;
   // GBK_TO_UNICODE[26810] := 16#CEF5;
   // GBK_TO_UNICODE[26811] := 16#7199;
   // GBK_TO_UNICODE[26812] := 16#CEF6;
   // GBK_TO_UNICODE[26813] := 16#6790;
   // GBK_TO_UNICODE[26814] := 16#CEF7;
   // GBK_TO_UNICODE[26815] := 16#897F;
   // GBK_TO_UNICODE[26816] := 16#CEF8;
   // GBK_TO_UNICODE[26817] := 16#7852;
   // GBK_TO_UNICODE[26818] := 16#CEF9;
   // GBK_TO_UNICODE[26819] := 16#77FD;
   // GBK_TO_UNICODE[26820] := 16#CEFA;
   // GBK_TO_UNICODE[26821] := 16#6670;
   // GBK_TO_UNICODE[26822] := 16#CEFB;
   // GBK_TO_UNICODE[26823] := 16#563B;
   // GBK_TO_UNICODE[26824] := 16#CEFC;
   // GBK_TO_UNICODE[26825] := 16#5438;
   // GBK_TO_UNICODE[26826] := 16#CEFD;
   // GBK_TO_UNICODE[26827] := 16#9521;
   // GBK_TO_UNICODE[26828] := 16#CEFE;
   // GBK_TO_UNICODE[26829] := 16#727A;
   // GBK_TO_UNICODE[26830] := 16#CF40;
   // GBK_TO_UNICODE[26831] := 16#87A5;
   // GBK_TO_UNICODE[26832] := 16#CF41;
   // GBK_TO_UNICODE[26833] := 16#87A6;
   // GBK_TO_UNICODE[26834] := 16#CF42;
   // GBK_TO_UNICODE[26835] := 16#87A7;
   // GBK_TO_UNICODE[26836] := 16#CF43;
   // GBK_TO_UNICODE[26837] := 16#87A9;
   // GBK_TO_UNICODE[26838] := 16#CF44;
   // GBK_TO_UNICODE[26839] := 16#87AA;
   // GBK_TO_UNICODE[26840] := 16#CF45;
   // GBK_TO_UNICODE[26841] := 16#87AE;
   // GBK_TO_UNICODE[26842] := 16#CF46;
   // GBK_TO_UNICODE[26843] := 16#87B0;
   // GBK_TO_UNICODE[26844] := 16#CF47;
   // GBK_TO_UNICODE[26845] := 16#87B1;
   // GBK_TO_UNICODE[26846] := 16#CF48;
   // GBK_TO_UNICODE[26847] := 16#87B2;
   // GBK_TO_UNICODE[26848] := 16#CF49;
   // GBK_TO_UNICODE[26849] := 16#87B4;
   // GBK_TO_UNICODE[26850] := 16#CF4A;
   // GBK_TO_UNICODE[26851] := 16#87B6;
   // GBK_TO_UNICODE[26852] := 16#CF4B;
   // GBK_TO_UNICODE[26853] := 16#87B7;
   // GBK_TO_UNICODE[26854] := 16#CF4C;
   // GBK_TO_UNICODE[26855] := 16#87B8;
   // GBK_TO_UNICODE[26856] := 16#CF4D;
   // GBK_TO_UNICODE[26857] := 16#87B9;
   // GBK_TO_UNICODE[26858] := 16#CF4E;
   // GBK_TO_UNICODE[26859] := 16#87BB;
   // GBK_TO_UNICODE[26860] := 16#CF4F;
   // GBK_TO_UNICODE[26861] := 16#87BC;
   // GBK_TO_UNICODE[26862] := 16#CF50;
   // GBK_TO_UNICODE[26863] := 16#87BE;
   // GBK_TO_UNICODE[26864] := 16#CF51;
   // GBK_TO_UNICODE[26865] := 16#87BF;
   // GBK_TO_UNICODE[26866] := 16#CF52;
   // GBK_TO_UNICODE[26867] := 16#87C1;
   // GBK_TO_UNICODE[26868] := 16#CF53;
   // GBK_TO_UNICODE[26869] := 16#87C2;
   // GBK_TO_UNICODE[26870] := 16#CF54;
   // GBK_TO_UNICODE[26871] := 16#87C3;
   // GBK_TO_UNICODE[26872] := 16#CF55;
   // GBK_TO_UNICODE[26873] := 16#87C4;
   // GBK_TO_UNICODE[26874] := 16#CF56;
   // GBK_TO_UNICODE[26875] := 16#87C5;
   // GBK_TO_UNICODE[26876] := 16#CF57;
   // GBK_TO_UNICODE[26877] := 16#87C7;
   // GBK_TO_UNICODE[26878] := 16#CF58;
   // GBK_TO_UNICODE[26879] := 16#87C8;
   // GBK_TO_UNICODE[26880] := 16#CF59;
   // GBK_TO_UNICODE[26881] := 16#87C9;
   // GBK_TO_UNICODE[26882] := 16#CF5A;
   // GBK_TO_UNICODE[26883] := 16#87CC;
   // GBK_TO_UNICODE[26884] := 16#CF5B;
   // GBK_TO_UNICODE[26885] := 16#87CD;
   // GBK_TO_UNICODE[26886] := 16#CF5C;
   // GBK_TO_UNICODE[26887] := 16#87CE;
   // GBK_TO_UNICODE[26888] := 16#CF5D;
   // GBK_TO_UNICODE[26889] := 16#87CF;
   // GBK_TO_UNICODE[26890] := 16#CF5E;
   // GBK_TO_UNICODE[26891] := 16#87D0;
   // GBK_TO_UNICODE[26892] := 16#CF5F;
   // GBK_TO_UNICODE[26893] := 16#87D4;
   // GBK_TO_UNICODE[26894] := 16#CF60;
   // GBK_TO_UNICODE[26895] := 16#87D5;
   // GBK_TO_UNICODE[26896] := 16#CF61;
   // GBK_TO_UNICODE[26897] := 16#87D6;
   // GBK_TO_UNICODE[26898] := 16#CF62;
   // GBK_TO_UNICODE[26899] := 16#87D7;
   // GBK_TO_UNICODE[26900] := 16#CF63;
   // GBK_TO_UNICODE[26901] := 16#87D8;
   // GBK_TO_UNICODE[26902] := 16#CF64;
   // GBK_TO_UNICODE[26903] := 16#87D9;
   // GBK_TO_UNICODE[26904] := 16#CF65;
   // GBK_TO_UNICODE[26905] := 16#87DA;
   // GBK_TO_UNICODE[26906] := 16#CF66;
   // GBK_TO_UNICODE[26907] := 16#87DC;
   // GBK_TO_UNICODE[26908] := 16#CF67;
   // GBK_TO_UNICODE[26909] := 16#87DD;
   // GBK_TO_UNICODE[26910] := 16#CF68;
   // GBK_TO_UNICODE[26911] := 16#87DE;
   // GBK_TO_UNICODE[26912] := 16#CF69;
   // GBK_TO_UNICODE[26913] := 16#87DF;
   // GBK_TO_UNICODE[26914] := 16#CF6A;
   // GBK_TO_UNICODE[26915] := 16#87E1;
   // GBK_TO_UNICODE[26916] := 16#CF6B;
   // GBK_TO_UNICODE[26917] := 16#87E2;
   // GBK_TO_UNICODE[26918] := 16#CF6C;
   // GBK_TO_UNICODE[26919] := 16#87E3;
   // GBK_TO_UNICODE[26920] := 16#CF6D;
   // GBK_TO_UNICODE[26921] := 16#87E4;
   // GBK_TO_UNICODE[26922] := 16#CF6E;
   // GBK_TO_UNICODE[26923] := 16#87E6;
   // GBK_TO_UNICODE[26924] := 16#CF6F;
   // GBK_TO_UNICODE[26925] := 16#87E7;
   // GBK_TO_UNICODE[26926] := 16#CF70;
   // GBK_TO_UNICODE[26927] := 16#87E8;
   // GBK_TO_UNICODE[26928] := 16#CF71;
   // GBK_TO_UNICODE[26929] := 16#87E9;
   // GBK_TO_UNICODE[26930] := 16#CF72;
   // GBK_TO_UNICODE[26931] := 16#87EB;
   // GBK_TO_UNICODE[26932] := 16#CF73;
   // GBK_TO_UNICODE[26933] := 16#87EC;
   // GBK_TO_UNICODE[26934] := 16#CF74;
   // GBK_TO_UNICODE[26935] := 16#87ED;
   // GBK_TO_UNICODE[26936] := 16#CF75;
   // GBK_TO_UNICODE[26937] := 16#87EF;
   // GBK_TO_UNICODE[26938] := 16#CF76;
   // GBK_TO_UNICODE[26939] := 16#87F0;
   // GBK_TO_UNICODE[26940] := 16#CF77;
   // GBK_TO_UNICODE[26941] := 16#87F1;
   // GBK_TO_UNICODE[26942] := 16#CF78;
   // GBK_TO_UNICODE[26943] := 16#87F2;
   // GBK_TO_UNICODE[26944] := 16#CF79;
   // GBK_TO_UNICODE[26945] := 16#87F3;
   // GBK_TO_UNICODE[26946] := 16#CF7A;
   // GBK_TO_UNICODE[26947] := 16#87F4;
   // GBK_TO_UNICODE[26948] := 16#CF7B;
   // GBK_TO_UNICODE[26949] := 16#87F5;
   // GBK_TO_UNICODE[26950] := 16#CF7C;
   // GBK_TO_UNICODE[26951] := 16#87F6;
   // GBK_TO_UNICODE[26952] := 16#CF7D;
   // GBK_TO_UNICODE[26953] := 16#87F7;
   // GBK_TO_UNICODE[26954] := 16#CF7E;
   // GBK_TO_UNICODE[26955] := 16#87F8;
   // GBK_TO_UNICODE[26956] := 16#CF80;
   // GBK_TO_UNICODE[26957] := 16#87FA;
   // GBK_TO_UNICODE[26958] := 16#CF81;
   // GBK_TO_UNICODE[26959] := 16#87FB;
   // GBK_TO_UNICODE[26960] := 16#CF82;
   // GBK_TO_UNICODE[26961] := 16#87FC;
   // GBK_TO_UNICODE[26962] := 16#CF83;
   // GBK_TO_UNICODE[26963] := 16#87FD;
   // GBK_TO_UNICODE[26964] := 16#CF84;
   // GBK_TO_UNICODE[26965] := 16#87FF;
   // GBK_TO_UNICODE[26966] := 16#CF85;
   // GBK_TO_UNICODE[26967] := 16#8800;
   // GBK_TO_UNICODE[26968] := 16#CF86;
   // GBK_TO_UNICODE[26969] := 16#8801;
   // GBK_TO_UNICODE[26970] := 16#CF87;
   // GBK_TO_UNICODE[26971] := 16#8802;
   // GBK_TO_UNICODE[26972] := 16#CF88;
   // GBK_TO_UNICODE[26973] := 16#8804;
   // GBK_TO_UNICODE[26974] := 16#CF89;
   // GBK_TO_UNICODE[26975] := 16#8805;
   // GBK_TO_UNICODE[26976] := 16#CF8A;
   // GBK_TO_UNICODE[26977] := 16#8806;
   // GBK_TO_UNICODE[26978] := 16#CF8B;
   // GBK_TO_UNICODE[26979] := 16#8807;
   // GBK_TO_UNICODE[26980] := 16#CF8C;
   // GBK_TO_UNICODE[26981] := 16#8808;
   // GBK_TO_UNICODE[26982] := 16#CF8D;
   // GBK_TO_UNICODE[26983] := 16#8809;
   // GBK_TO_UNICODE[26984] := 16#CF8E;
   // GBK_TO_UNICODE[26985] := 16#880B;
   // GBK_TO_UNICODE[26986] := 16#CF8F;
   // GBK_TO_UNICODE[26987] := 16#880C;
   // GBK_TO_UNICODE[26988] := 16#CF90;
   // GBK_TO_UNICODE[26989] := 16#880D;
   // GBK_TO_UNICODE[26990] := 16#CF91;
   // GBK_TO_UNICODE[26991] := 16#880E;
   // GBK_TO_UNICODE[26992] := 16#CF92;
   // GBK_TO_UNICODE[26993] := 16#880F;
   // GBK_TO_UNICODE[26994] := 16#CF93;
   // GBK_TO_UNICODE[26995] := 16#8810;
   // GBK_TO_UNICODE[26996] := 16#CF94;
   // GBK_TO_UNICODE[26997] := 16#8811;
   // GBK_TO_UNICODE[26998] := 16#CF95;
   // GBK_TO_UNICODE[26999] := 16#8812;
   // GBK_TO_UNICODE[27000] := 16#CF96;
   // GBK_TO_UNICODE[27001] := 16#8814;
   // GBK_TO_UNICODE[27002] := 16#CF97;
   // GBK_TO_UNICODE[27003] := 16#8817;
   // GBK_TO_UNICODE[27004] := 16#CF98;
   // GBK_TO_UNICODE[27005] := 16#8818;
   // GBK_TO_UNICODE[27006] := 16#CF99;
   // GBK_TO_UNICODE[27007] := 16#8819;
   // GBK_TO_UNICODE[27008] := 16#CF9A;
   // GBK_TO_UNICODE[27009] := 16#881A;
   // GBK_TO_UNICODE[27010] := 16#CF9B;
   // GBK_TO_UNICODE[27011] := 16#881C;
   // GBK_TO_UNICODE[27012] := 16#CF9C;
   // GBK_TO_UNICODE[27013] := 16#881D;
   // GBK_TO_UNICODE[27014] := 16#CF9D;
   // GBK_TO_UNICODE[27015] := 16#881E;
   // GBK_TO_UNICODE[27016] := 16#CF9E;
   // GBK_TO_UNICODE[27017] := 16#881F;
   // GBK_TO_UNICODE[27018] := 16#CF9F;
   // GBK_TO_UNICODE[27019] := 16#8820;
   // GBK_TO_UNICODE[27020] := 16#CFA0;
   // GBK_TO_UNICODE[27021] := 16#8823;
   // GBK_TO_UNICODE[27022] := 16#CFA1;
   // GBK_TO_UNICODE[27023] := 16#7A00;
   // GBK_TO_UNICODE[27024] := 16#CFA2;
   // GBK_TO_UNICODE[27025] := 16#606F;
   // GBK_TO_UNICODE[27026] := 16#CFA3;
   // GBK_TO_UNICODE[27027] := 16#5E0C;
   // GBK_TO_UNICODE[27028] := 16#CFA4;
   // GBK_TO_UNICODE[27029] := 16#6089;
   // GBK_TO_UNICODE[27030] := 16#CFA5;
   // GBK_TO_UNICODE[27031] := 16#819D;
   // GBK_TO_UNICODE[27032] := 16#CFA6;
   // GBK_TO_UNICODE[27033] := 16#5915;
   // GBK_TO_UNICODE[27034] := 16#CFA7;
   // GBK_TO_UNICODE[27035] := 16#60DC;
   // GBK_TO_UNICODE[27036] := 16#CFA8;
   // GBK_TO_UNICODE[27037] := 16#7184;
   // GBK_TO_UNICODE[27038] := 16#CFA9;
   // GBK_TO_UNICODE[27039] := 16#70EF;
   // GBK_TO_UNICODE[27040] := 16#CFAA;
   // GBK_TO_UNICODE[27041] := 16#6EAA;
   // GBK_TO_UNICODE[27042] := 16#CFAB;
   // GBK_TO_UNICODE[27043] := 16#6C50;
   // GBK_TO_UNICODE[27044] := 16#CFAC;
   // GBK_TO_UNICODE[27045] := 16#7280;
   // GBK_TO_UNICODE[27046] := 16#CFAD;
   // GBK_TO_UNICODE[27047] := 16#6A84;
   // GBK_TO_UNICODE[27048] := 16#CFAE;
   // GBK_TO_UNICODE[27049] := 16#88AD;
   // GBK_TO_UNICODE[27050] := 16#CFAF;
   // GBK_TO_UNICODE[27051] := 16#5E2D;
   // GBK_TO_UNICODE[27052] := 16#CFB0;
   // GBK_TO_UNICODE[27053] := 16#4E60;
   // GBK_TO_UNICODE[27054] := 16#CFB1;
   // GBK_TO_UNICODE[27055] := 16#5AB3;
   // GBK_TO_UNICODE[27056] := 16#CFB2;
   // GBK_TO_UNICODE[27057] := 16#559C;
   // GBK_TO_UNICODE[27058] := 16#CFB3;
   // GBK_TO_UNICODE[27059] := 16#94E3;
   // GBK_TO_UNICODE[27060] := 16#CFB4;
   // GBK_TO_UNICODE[27061] := 16#6D17;
   // GBK_TO_UNICODE[27062] := 16#CFB5;
   // GBK_TO_UNICODE[27063] := 16#7CFB;
   // GBK_TO_UNICODE[27064] := 16#CFB6;
   // GBK_TO_UNICODE[27065] := 16#9699;
   // GBK_TO_UNICODE[27066] := 16#CFB7;
   // GBK_TO_UNICODE[27067] := 16#620F;
